                        IF temporalCounter_i1.done THEN 
                            (* Transition: '<S30>:42' *)
                            is_c47_ChiefMaster := ChiefMaster_IN_Error;
                            (* Entry 'Error': '<S30>:38' *)
                            (* '<S30>:38:2' MainHV_Minus_Welded = true *)
                            MainHV_Minus_Welded := TRUE;
                            (* '<S30>:38:3' MainHV_Plus_Welded = true *)
                            MainHV_Plus_Welded := TRUE;
                            (* '<S30>:38:4' WeldingDetection_Status = uint8(2); *)
                            WeldingDetection_Status := 2;
                        ELSE 
                            (* '<S30>:40:2' REQ_MainHV_ON_PLUS = false *)
                            REQ_MainHV_ON_PLUS := FALSE;
                            (* '<S30>:40:3' REQ_MainHV_ON_MINUS = false *)
                            REQ_MainHV_ON_MINUS := FALSE;
                            (* '<S30>:40:4' MainHV_Minus_Welded = false *)
                            MainHV_Minus_Welded := FALSE;
                            (* '<S30>:40:5' MainHV_Plus_Welded = false *)
                            MainHV_Plus_Welded := FALSE;
                        END_IF;

                    END_IF;

                ChiefMaster_IN_Open1: 
                    (* During 'Open1': '<S30>:28' *)
                    (* '<S30>:44:1' sf_internal_predicateOutput = In == true; *)

                    IF In THEN 
                        (* Transition: '<S30>:44' *)
                        is_c47_ChiefMaster := b_ChiefMaster_IN_Open;
                        temporalCounter_i1(timerAction := 1, maxTime := 0);
                        (* Entry 'Open': '<S30>:40' *)
                        (* '<S30>:40:2' REQ_MainHV_ON_PLUS = false *)
                        REQ_MainHV_ON_PLUS := FALSE;
                        (* '<S30>:40:3' REQ_MainHV_ON_MINUS = false *)
                        REQ_MainHV_ON_MINUS := FALSE;
                        (* '<S30>:40:4' MainHV_Minus_Welded = false *)
                        MainHV_Minus_Welded := FALSE;
                        (* '<S30>:40:5' MainHV_Plus_Welded = false *)
                        MainHV_Plus_Welded := FALSE;
                    ELSE 
                        (* '<S30>:28:2' REQ_MainHV_ON_PLUS = false *)
                        REQ_MainHV_ON_PLUS := FALSE;
                        (* '<S30>:28:3' REQ_MainHV_ON_MINUS = false *)
                        REQ_MainHV_ON_MINUS := FALSE;
                        (* '<S30>:28:4' MainHV_Minus_Welded = false *)
                        MainHV_Minus_Welded := FALSE;
                        (* '<S30>:28:5' MainHV_Plus_Welded = false *)
                        MainHV_Plus_Welded := FALSE;
                        (* '<S30>:28:6' WeldingDetection_Status = uint8(1); *)
                        WeldingDetection_Status := 1;
                    END_IF;

                ELSE
                    (* During 'Plus_Close': '<S30>:4' *)
                    (* '<S30>:13:1' sf_internal_predicateOutput = LoadVtg <= 20; *)

                    IF LoadVtg <= 20.0 THEN 
                        (* Transition: '<S30>:13' *)
                        is_c47_ChiefMaster := ChiefMaster_IN_Minus_Close;
                        temporalCounter_i1(timerAction := 1, maxTime := 0);
                        (* Entry 'Minus_Close': '<S30>:12' *)
                        (* '<S30>:12:2' REQ_MainHV_ON_MINUS = true *)
                        REQ_MainHV_ON_MINUS := TRUE;
                    ELSE 
                        (* '<S30>:23:1' sf_internal_predicateOutput = after(5,sec); *)
                        temporalCounter_i1(timerAction := 2, maxTime := 5000);

                        IF temporalCounter_i1.done THEN 
                            (* Transition: '<S30>:23' *)
                            is_c47_ChiefMaster := ChiefMaster_IN_ErrorMinus;
                            (* Entry 'ErrorMinus': '<S30>:22' *)
                            (* '<S30>:22:2' MainHV_Minus_Welded = true *)
                            MainHV_Minus_Welded := TRUE;
                            (* '<S30>:22:3' WeldingDetection_Status = uint8(2); *)
                            WeldingDetection_Status := 2;
                        ELSE 
                            (* '<S30>:4:2' REQ_MainHV_ON_PLUS = true *)
                            REQ_MainHV_ON_PLUS := TRUE;
                        END_IF;

                    END_IF;

            END_CASE;

        END_IF;

        (* End of Chart: '<S22>/Chart_WeldingDetection' *)
END_CASE;

END_FUNCTION_BLOCK

// Device/Application/Chart_jj
FUNCTION_BLOCK Chart_jj
VAR_INPUT
	ssMethodType: SINT;
	In: LREAL;
	b_n: LREAL;
END_VAR
VAR_OUTPUT
	Out: BOOL;
END_VAR
VAR
	temporalCounter_i1: PLC_CODER_TIMER;
	is_c10_ChiefMaster: USINT;
	is_active_c10_ChiefMaster: USINT;
END_VAR



CASE ssMethodType OF
    SS_INITIALIZE: 
        temporalCounter_i1(timerAction := 1, maxTime := 0);
        is_active_c10_ChiefMaster := 0;
        is_c10_ChiefMaster := ChiefMaster_IN_NO_ACTIVE_CHILD_a4;
        Out := FALSE;
    SS_OUTPUT: 
        (* Chart: '<S81>/Chart' *)
        (* Gateway: ChiefMaster/Flow Logic/Reset/Reset_Req/Subsystem1/Chart *)
        (* During: ChiefMaster/Flow Logic/Reset/Reset_Req/Subsystem1/Chart *)

        IF is_active_c10_ChiefMaster = 0 THEN 
            (* Entry: ChiefMaster/Flow Logic/Reset/Reset_Req/Subsystem1/Chart *)
            is_active_c10_ChiefMaster := 1;
            (* Entry Internal: ChiefMaster/Flow Logic/Reset/Reset_Req/Subsystem1/Chart *)
            (* Transition: '<S87>:3' *)
            is_c10_ChiefMaster := ChiefMaster_IN_Default_m;
            (* Entry 'Default': '<S87>:2' *)
            (* '<S87>:2:2' Out = false *)
            Out := FALSE;
        ELSE 

            CASE is_c10_ChiefMaster OF
                ChiefMaster_IN_Default_m: 
                    (* During 'Default': '<S87>:2' *)
                    (* '<S87>:6:1' sf_internal_predicateOutput = In == 2; *)

                    IF In = 2.0 THEN 
                        (* Transition: '<S87>:6' *)
                        is_c10_ChiefMaster := ChiefMaster_IN_Delay;
                        temporalCounter_i1(timerAction := 1, maxTime := 0);
                        (* Entry 'Delay': '<S87>:5' *)
                        (* '<S87>:5:2' Out = false *)
                        Out := FALSE;
                    ELSE 
                        (* '<S87>:2:2' Out = false *)
                        Out := FALSE;
                    END_IF;

                ChiefMaster_IN_Delay: 
                    (* During 'Delay': '<S87>:5' *)
                    (* '<S87>:12:1' sf_internal_predicateOutput = after(n,sec); *)
                    temporalCounter_i1(timerAction := 2, maxTime := TRUNC(b_n * 1000.0));

                    IF temporalCounter_i1.done THEN 
                        (* Transition: '<S87>:12' *)
                        is_c10_ChiefMaster := b_ChiefMaster_IN_Delay1;
                        (* Entry 'Delay1': '<S87>:11' *)
                        (* '<S87>:11:2' Out = true *)
                        Out := TRUE;
                    ELSE 
                        (* '<S87>:13:1' sf_internal_predicateOutput = In == 1 ||... *)
                        (* '<S87>:13:2' In == 3; *)

                        IF (In = 1.0) OR (In = 3.0) THEN 
                            (* Transition: '<S87>:13' *)
                            is_c10_ChiefMaster := ChiefMaster_IN_Default_m;
                            (* Entry 'Default': '<S87>:2' *)
                            (* '<S87>:2:2' Out = false *)
                            Out := FALSE;
                        ELSE 
                            (* '<S87>:5:2' Out = false *)
                            Out := FALSE;
                        END_IF;

                    END_IF;

                ELSE
                    (* During 'Delay1': '<S87>:11' *)
                    (* '<S87>:14:1' sf_internal_predicateOutput = In == 3; *)

                    IF In = 3.0 THEN 
                        (* Transition: '<S87>:14' *)
                        is_c10_ChiefMaster := ChiefMaster_IN_Default_m;
                        (* Entry 'Default': '<S87>:2' *)
                        (* '<S87>:2:2' Out = false *)
                        Out := FALSE;
                    ELSE 
                        (* '<S87>:11:2' Out = true *)
                        Out := TRUE;
                    END_IF;

            END_CASE;

        END_IF;

        (* End of Chart: '<S81>/Chart' *)
END_CASE;

END_FUNCTION_BLOCK

// Device/Application/Chart1
FUNCTION_BLOCK Chart1
VAR_INPUT
	ssMethodType: SINT;
	In: BOOL;
END_VAR
VAR_OUTPUT
	Out: BOOL;
END_VAR
VAR
	is_active_c12_ChiefMaster: USINT;
	is_c12_ChiefMaster: USINT;
	temporalCounter_i1: PLC_CODER_TIMER;
END_VAR



CASE ssMethodType OF
    SS_INITIALIZE: 
        temporalCounter_i1(timerAction := 1, maxTime := 0);
        is_active_c12_ChiefMaster := 0;
        is_c12_ChiefMaster := ChiefMaster_IN_NO_ACTIVE_CHILD_kt;
        Out := FALSE;
    SS_OUTPUT: 
        (* Chart: '<S81>/Chart1' *)
        (* Gateway: ChiefMaster/Flow Logic/Reset/Reset_Req/Subsystem1/Chart1 *)
        (* During: ChiefMaster/Flow Logic/Reset/Reset_Req/Subsystem1/Chart1 *)

        IF is_active_c12_ChiefMaster = 0 THEN 
            (* Entry: ChiefMaster/Flow Logic/Reset/Reset_Req/Subsystem1/Chart1 *)
            is_active_c12_ChiefMaster := 1;
            (* Entry Internal: ChiefMaster/Flow Logic/Reset/Reset_Req/Subsystem1/Chart1 *)
            (* Transition: '<S88>:3' *)
            is_c12_ChiefMaster := ChiefMaster_IN_Default_dh;
            (* Entry 'Default': '<S88>:2' *)
            (* '<S88>:2:2' Out = false *)
            Out := FALSE;
        ELSE 

            CASE is_c12_ChiefMaster OF
                ChiefMaster_IN_Default_dh: 
                    (* During 'Default': '<S88>:2' *)
                    (* '<S88>:6:1' sf_internal_predicateOutput = In == true; *)

                    IF In THEN 
                        (* Transition: '<S88>:6' *)
                        is_c12_ChiefMaster := ChiefMaster_IN_Delay_j;
                        temporalCounter_i1(timerAction := 1, maxTime := 0);
                        (* Entry 'Delay': '<S88>:5' *)
                        (* '<S88>:5:2' Out = true *)
                        Out := TRUE;
                    ELSE 
                        (* '<S88>:2:2' Out = false *)
                        Out := FALSE;
                    END_IF;

                ChiefMaster_IN_Delay_j: 
                    (* During 'Delay': '<S88>:5' *)
                    (* '<S88>:21:1' sf_internal_predicateOutput = after(10,msec); *)
                    temporalCounter_i1(timerAction := 2, maxTime := 10);

                    IF temporalCounter_i1.done THEN 
                        (* Transition: '<S88>:21' *)
                        is_c12_ChiefMaster := ChiefMaster_IN_pulse;
                        (* Entry 'pulse': '<S88>:20' *)
                        (* '<S88>:20:2' Out = false *)
                        Out := FALSE;
                    ELSE 
                        (* '<S88>:5:2' Out = true *)
                        Out := TRUE;
                    END_IF;

                ELSE
                    (* During 'pulse': '<S88>:20' *)
                    (* '<S88>:20:2' Out = false *)
                    Out := FALSE;
            END_CASE;

        END_IF;

        (* End of Chart: '<S81>/Chart1' *)
END_CASE;

END_FUNCTION_BLOCK

// Device/Application/Chart_lg
FUNCTION_BLOCK Chart_lg
VAR_INPUT
	ssMethodType: SINT;
	Error: BOOL;
	KL15_reset: BOOL;
END_VAR
VAR_OUTPUT
	SW_Reset: BOOL;
END_VAR
VAR
	temporalCounter_i1: PLC_CODER_TIMER;
	is_c13_ChiefMaster: USINT;
	is_active_c13_ChiefMaster: USINT;
END_VAR



CASE ssMethodType OF
    SS_INITIALIZE: 
        temporalCounter_i1(timerAction := 1, maxTime := 0);
        is_active_c13_ChiefMaster := 0;
        is_c13_ChiefMaster := ChiefMaster_IN_NO_ACTIVE_CHILD_a0;
        SW_Reset := FALSE;
    SS_OUTPUT: 
        (* Chart: '<S83>/Chart' *)
        (* Gateway: ChiefMaster/Flow Logic/Reset/Reset_Req/Subsystem3/Chart *)
        (* During: ChiefMaster/Flow Logic/Reset/Reset_Req/Subsystem3/Chart *)

        IF is_active_c13_ChiefMaster = 0 THEN 
            (* Entry: ChiefMaster/Flow Logic/Reset/Reset_Req/Subsystem3/Chart *)
            is_active_c13_ChiefMaster := 1;
            (* Entry Internal: ChiefMaster/Flow Logic/Reset/Reset_Req/Subsystem3/Chart *)
            (* Transition: '<S91>:3' *)
            is_c13_ChiefMaster := ChiefMaster_IN_Default_e0;
            (* Entry 'Default': '<S91>:2' *)
            (* '<S91>:2:2' SW_Reset = false *)
            SW_Reset := FALSE;
        ELSE 

            CASE is_c13_ChiefMaster OF
                ChiefMaster_IN_Default_e0: 
                    (* During 'Default': '<S91>:2' *)
                    (* '<S91>:6:1' sf_internal_predicateOutput = Error == true; *)

                    IF Error THEN 
                        (* Transition: '<S91>:6' *)
                        is_c13_ChiefMaster := ChiefMaster_IN_hold_hw;
                        temporalCounter_i1(timerAction := 1, maxTime := 0);
                        (* Entry 'hold': '<S91>:5' *)
                        (* '<S91>:5:2' SW_Reset = false *)
                        SW_Reset := FALSE;
                    ELSE 
                        (* '<S91>:2:2' SW_Reset = false *)
                        SW_Reset := FALSE;
                    END_IF;

                ChiefMaster_IN_Delay_i: 
                    (* During 'Delay': '<S91>:11' *)
                    (* '<S91>:16:1' sf_internal_predicateOutput = after(10,msec); *)
                    temporalCounter_i1(timerAction := 2, maxTime := 10);

                    IF temporalCounter_i1.done THEN 
                        (* Transition: '<S91>:16' *)
                        is_c13_ChiefMaster := ChiefMaster_IN_pulse_i;
                        (* Entry 'pulse': '<S91>:15' *)
                        (* '<S91>:15:2' SW_Reset = false *)
                        SW_Reset := FALSE;
                    ELSE 
                        (* '<S91>:11:2' SW_Reset = true *)
                        SW_Reset := TRUE;
                    END_IF;

                ChiefMaster_IN_KL15_reset: 
                    (* During 'KL15_reset': '<S91>:18' *)
                    (* '<S91>:21:1' sf_internal_predicateOutput = after(25,sec) &&... *)
                    (* '<S91>:21:2' Error == false; *)
                    temporalCounter_i1(timerAction := 2, maxTime := 25000);

                    IF temporalCounter_i1.done THEN 

                        IF  NOT Error THEN 
                            (* Transition: '<S91>:21' *)
                            is_c13_ChiefMaster := ChiefMaster_IN_Default_e0;
                            (* Entry 'Default': '<S91>:2' *)
                            (* '<S91>:2:2' SW_Reset = false *)
                            SW_Reset := FALSE;
                        ELSE 
                            (* '<S91>:18:2' SW_Reset = false *)
                            SW_Reset := FALSE;
                        END_IF;

                    ELSE 
                        (* '<S91>:18:2' SW_Reset = false *)
                        SW_Reset := FALSE;
                    END_IF;

                ChiefMaster_IN_hold_hw: 
                    (* During 'hold': '<S91>:5' *)
                    (* '<S91>:12:1' sf_internal_predicateOutput = after(5,sec); *)
                    temporalCounter_i1(timerAction := 2, maxTime := 5000);

                    IF temporalCounter_i1.done THEN 
                        (* Transition: '<S91>:12' *)
                        is_c13_ChiefMaster := ChiefMaster_IN_Delay_i;
                        temporalCounter_i1(timerAction := 1, maxTime := 0);
                        (* Entry 'Delay': '<S91>:11' *)
                        (* '<S91>:11:2' SW_Reset = true *)
                        SW_Reset := TRUE;
                    ELSE 
                        (* '<S91>:13:1' sf_internal_predicateOutput = Error == false; *)

                        IF  NOT Error THEN 
                            (* Transition: '<S91>:13' *)
                            is_c13_ChiefMaster := ChiefMaster_IN_Default_e0;
                            (* Entry 'Default': '<S91>:2' *)
                            (* '<S91>:2:2' SW_Reset = false *)
                            SW_Reset := FALSE;
                        ELSE 
                            (* '<S91>:5:2' SW_Reset = false *)
                            SW_Reset := FALSE;
                        END_IF;

                    END_IF;

                ELSE
                    (* During 'pulse': '<S91>:15' *)
                    (* '<S91>:17:1' sf_internal_predicateOutput = KL15_reset == true; *)

                    IF KL15_reset THEN 
                        (* Transition: '<S91>:17' *)
                        is_c13_ChiefMaster := ChiefMaster_IN_KL15_reset;
                        temporalCounter_i1(timerAction := 1, maxTime := 0);
                        (* Entry 'KL15_reset': '<S91>:18' *)
                        (* '<S91>:18:2' SW_Reset = false *)
                        SW_Reset := FALSE;
                    ELSE 
                        (* '<S91>:15:2' SW_Reset = false *)
                        SW_Reset := FALSE;
                    END_IF;

            END_CASE;

        END_IF;

        (* End of Chart: '<S83>/Chart' *)
END_CASE;

END_FUNCTION_BLOCK

// Device/Application/Chart1_l
FUNCTION_BLOCK Chart1_l
VAR_INPUT
	ssMethodType: SINT;
	SW_Reset: BOOL;
	KL_15_reset_CM: BOOL;
END_VAR
VAR_OUTPUT
	Count: LREAL;
END_VAR
VAR
	is_active_c14_ChiefMaster: USINT;
	is_c14_ChiefMaster: USINT;
END_VAR



CASE ssMethodType OF
    SS_INITIALIZE: 
        is_active_c14_ChiefMaster := 0;
        is_c14_ChiefMaster := ChiefMaster_IN_NO_ACTIVE_CHILD_a1;
        Count := 0.0;
    SS_OUTPUT: 
        (* Chart: '<S83>/Chart1' *)
        (* Gateway: ChiefMaster/Flow Logic/Reset/Reset_Req/Subsystem3/Chart1 *)
        (* During: ChiefMaster/Flow Logic/Reset/Reset_Req/Subsystem3/Chart1 *)

        IF is_active_c14_ChiefMaster = 0 THEN 
            (* Entry: ChiefMaster/Flow Logic/Reset/Reset_Req/Subsystem3/Chart1 *)
            is_active_c14_ChiefMaster := 1;
            (* Entry Internal: ChiefMaster/Flow Logic/Reset/Reset_Req/Subsystem3/Chart1 *)
            (* Transition: '<S92>:3' *)
            is_c14_ChiefMaster := ChiefMaster_IN_Default_g;
            (* Entry 'Default': '<S92>:2' *)
            (* '<S92>:2:2' Count = 0 *)
            Count := 0.0;
        ELSE 

            CASE is_c14_ChiefMaster OF
                ChiefMaster_IN_Default_g: 
                    (* During 'Default': '<S92>:2' *)
                    (* '<S92>:6:1' sf_internal_predicateOutput = SW_Reset == true; *)

                    IF SW_Reset THEN 
                        (* Transition: '<S92>:6' *)
                        is_c14_ChiefMaster := ChiefMaster_IN_Delay_m;
                        (* Entry 'Delay': '<S92>:5' *)
                        (* '<S92>:5:2' Count = Count + 1 *)
                        Count := Count + 1.0;
                    ELSE 
                        (* '<S92>:2:2' Count = 0 *)
                        Count := 0.0;
                    END_IF;

                ChiefMaster_IN_Delay_m: 
                    (* During 'Delay': '<S92>:5' *)
                    (* '<S92>:28:1' sf_internal_predicateOutput = SW_Reset == false; *)

                    IF  NOT SW_Reset THEN 
                        (* Transition: '<S92>:28' *)
                        is_c14_ChiefMaster := ChiefMaster_IN_Delay1_h;
                        (* Entry 'Delay1': '<S92>:27' *)
                    ELSE 
                        (* '<S92>:5:2' Count = Count + 1 *)
                        Count := Count + 1.0;
                    END_IF;

                ELSE
                    (* During 'Delay1': '<S92>:27' *)
                    (* '<S92>:24:1' sf_internal_predicateOutput = KL_15_reset_CM == true; *)

                    IF KL_15_reset_CM THEN 
                        (* Transition: '<S92>:24' *)
                        is_c14_ChiefMaster := ChiefMaster_IN_Default_g;
                        (* Entry 'Default': '<S92>:2' *)
                        (* '<S92>:2:2' Count = 0 *)
                        Count := 0.0;
                    ELSE 
                        (* '<S92>:29:1' sf_internal_predicateOutput = SW_Reset == true; *)

                        IF SW_Reset THEN 
                            (* Transition: '<S92>:29' *)
                            is_c14_ChiefMaster := ChiefMaster_IN_Delay_m;
                            (* Entry 'Delay': '<S92>:5' *)
                            (* '<S92>:5:2' Count = Count + 1 *)
                            Count := Count + 1.0;
                        END_IF;

                    END_IF;

            END_CASE;

        END_IF;

        (* End of Chart: '<S83>/Chart1' *)
END_CASE;

END_FUNCTION_BLOCK

// Device/Application/CMState
FUNCTION_BLOCK CMState
VAR_INPUT
	ssMethodType: SINT;
	KL15: BOOL;
	KL15_AllBoxes: BOOL;
	InsulationReadyOK: BOOL;
	BattRelay_Closed: BOOL;
	IMD_Available: BOOL;
	BattRelay_Close_Req: BOOL;
	REQ_IMD_ON: BOOL;
	FL_boREQ_MainHV_ON_MINUS: BOOL;
	MainHV_Plus_Status: LREAL;
	ShutdownError: BOOL;
END_VAR
VAR_OUTPUT
	FL_u8SS_ChiefMaster_State: USINT;
END_VAR
VAR
	is_c27_ChiefMaster: USINT;
	is_active_c27_ChiefMaster: USINT;
	is_ON: USINT;
	is_OFF: USINT;
	tmp: BOOL;
END_VAR



CASE ssMethodType OF
    SS_INITIALIZE: 
        (* SystemInitialize for Chart: '<S109>/CMState' *)
        is_OFF := ChiefMaster_IN_NO_ACTIVE_CHILD_ktp;
        is_ON := ChiefMaster_IN_NO_ACTIVE_CHILD_ktp;
        is_active_c27_ChiefMaster := 0;
        is_c27_ChiefMaster := ChiefMaster_IN_NO_ACTIVE_CHILD_ktp;
        FL_u8SS_ChiefMaster_State := 0;
    SS_OUTPUT: 
        (* Chart: '<S109>/CMState' *)
        (* Gateway: ChiefMaster/Flow Logic/System Status/CMState/CMState *)
        (* During: ChiefMaster/Flow Logic/System Status/CMState/CMState *)

        IF is_active_c27_ChiefMaster = 0 THEN 
            (* Entry: ChiefMaster/Flow Logic/System Status/CMState/CMState *)
            is_active_c27_ChiefMaster := 1;
            (* Entry Internal: ChiefMaster/Flow Logic/System Status/CMState/CMState *)
            (* Transition: '<S124>:2' *)
            is_c27_ChiefMaster := ChiefMaster_IN_Sleep;
            (* Entry 'Sleep': '<S124>:1' *)
            (* '<S124>:1:2' CMState=0; *)
            FL_u8SS_ChiefMaster_State := 0;
        ELSE 

            CASE is_c27_ChiefMaster OF
                ChiefMaster_IN_Error_o: 
                    (* During 'Error': '<S124>:99' *)
                    (* '<S124>:116:1' sf_internal_predicateOutput = ShutdownError == false &&... *)
                    (* '<S124>:116:2' KL15==true; *)
                    tmp :=  NOT ShutdownError;

                    IF tmp AND KL15 THEN 
                        (* Transition: '<S124>:116' *)
                        is_c27_ChiefMaster := ChiefMaster_IN_ON;
                        (* Entry Internal 'ON': '<S124>:31' *)
                        (* Transition: '<S124>:62' *)
                        is_ON := ChiefMaster_IN_KL15ON;
                        (* Entry 'KL15ON': '<S124>:3' *)
                        (* '<S124>:3:2' CMState=1; *)
                        FL_u8SS_ChiefMaster_State := 1;
                    ELSE 
                        (* '<S124>:117:1' sf_internal_predicateOutput = ShutdownError == false &&... *)
                        (* '<S124>:117:2' KL15==false; *)

                        IF tmp AND ( NOT KL15) THEN 
                            (* Transition: '<S124>:117' *)
                            is_c27_ChiefMaster := ChiefMaster_IN_OFF;
                            (* Entry Internal 'OFF': '<S124>:90' *)
                            (* Transition: '<S124>:92' *)
                            is_OFF := ChiefMaster_IN_BDURelayOpen_Req;
                            (* Entry 'BDURelayOpen_Req': '<S124>:82' *)
                            (* '<S124>:82:2' CMState=8; *)
                            FL_u8SS_ChiefMaster_State := 8;
                        ELSE 
                            (* '<S124>:99:2' CMState=14; *)
                            FL_u8SS_ChiefMaster_State := 14;
                        END_IF;

                    END_IF;

                ChiefMaster_IN_OFF: 
                    (* During 'OFF': '<S124>:90' *)
                    (* '<S124>:96:1' sf_internal_predicateOutput = CMState==13; *)

                    IF FL_u8SS_ChiefMaster_State = 13 THEN 
                        (* Transition: '<S124>:96' *)
                        (* Exit Internal 'OFF': '<S124>:90' *)
                        is_OFF := ChiefMaster_IN_NO_ACTIVE_CHILD_ktp;
                        is_c27_ChiefMaster := ChiefMaster_IN_Sleep;
                        (* Entry 'Sleep': '<S124>:1' *)
                        (* '<S124>:1:2' CMState=0; *)
                        FL_u8SS_ChiefMaster_State := 0;
                    ELSE 
                        (* '<S124>:100:1' sf_internal_predicateOutput = ShutdownError == true; *)

                        IF ShutdownError THEN 
                            (* Transition: '<S124>:100' *)
                            (* Exit Internal 'OFF': '<S124>:90' *)
                            is_OFF := ChiefMaster_IN_NO_ACTIVE_CHILD_ktp;
                            is_c27_ChiefMaster := ChiefMaster_IN_Error_o;
                            (* Entry 'Error': '<S124>:99' *)
                            (* '<S124>:99:2' CMState=14; *)
                            FL_u8SS_ChiefMaster_State := 14;
                        ELSE 

                            CASE is_OFF OF
                                ChiefMaster_IN_BDURelayOpen: 
                                    (* During 'BDURelayOpen': '<S124>:86' *)
                                    (* '<S124>:84:1' sf_internal_predicateOutput = BattRelay_Close_Req==false; *)

                                    IF  NOT BattRelay_Close_Req THEN 
                                        (* Transition: '<S124>:84' *)
                                        is_OFF := ChiefMaster_IN_BattRelayOpen_Req;
                                        (* Entry 'BattRelayOpen_Req': '<S124>:94' *)
                                        (* '<S124>:94:2' CMState=10; *)
                                        FL_u8SS_ChiefMaster_State := 10;
                                    ELSE 
                                        (* '<S124>:86:2' CMState=9; *)
                                        FL_u8SS_ChiefMaster_State := 9;
                                    END_IF;

                                ChiefMaster_IN_BDURelayOpen_Req: 
                                    (* During 'BDURelayOpen_Req': '<S124>:82' *)
                                    (* '<S124>:93:1' sf_internal_predicateOutput = MainHV_Plus_Status==0; *)

                                    IF MainHV_Plus_Status = 0.0 THEN 
                                        (* Transition: '<S124>:93' *)
                                        is_OFF := ChiefMaster_IN_BDURelayOpen;
                                        (* Entry 'BDURelayOpen': '<S124>:86' *)
                                        (* '<S124>:86:2' CMState=9; *)
                                        FL_u8SS_ChiefMaster_State := 9;
                                    ELSE 
                                        (* '<S124>:82:2' CMState=8; *)
                                        FL_u8SS_ChiefMaster_State := 8;
                                    END_IF;

                                ChiefMaster_IN_BattRelayOpen: 
                                    (* During 'BattRelayOpen': '<S124>:89' *)
                                    (* '<S124>:83:1' sf_internal_predicateOutput = REQ_IMD_ON == false; *)

                                    IF  NOT REQ_IMD_ON THEN 
                                        (* Transition: '<S124>:83' *)
                                        is_OFF := ChiefMaster_IN_ISOMonitorOFF;
                                        (* Entry 'ISOMonitorOFF': '<S124>:88' *)
                                        (* '<S124>:88:2' CMState=12; *)
                                        FL_u8SS_ChiefMaster_State := 12;
                                    ELSE 
                                        (* '<S124>:89:2' CMState=11; *)
                                        FL_u8SS_ChiefMaster_State := 11;
                                    END_IF;

                                ChiefMaster_IN_BattRelayOpen_Req: 
                                    (* During 'BattRelayOpen_Req': '<S124>:94' *)
                                    (* '<S124>:95:1' sf_internal_predicateOutput = BattRelay_Closed==false; *)

                                    IF  NOT BattRelay_Closed THEN 
                                        (* Transition: '<S124>:95' *)
                                        is_OFF := ChiefMaster_IN_BattRelayOpen;
                                        (* Entry 'BattRelayOpen': '<S124>:89' *)
                                        (* '<S124>:89:2' CMState=11; *)
                                        FL_u8SS_ChiefMaster_State := 11;
                                    ELSE 
                                        (* '<S124>:94:2' CMState=10; *)
                                        FL_u8SS_ChiefMaster_State := 10;
                                    END_IF;

                                ChiefMaster_IN_ISOMonitorOFF: 
                                    (* During 'ISOMonitorOFF': '<S124>:88' *)
                                    (* '<S124>:85:1' sf_internal_predicateOutput = KL15_AllBoxes==false; *)

                                    IF  NOT KL15_AllBoxes THEN 
                                        (* Transition: '<S124>:85' *)
                                        is_OFF := ChiefMaster_IN_KL15OFF;
                                        (* Entry 'KL15OFF': '<S124>:91' *)
                                        (* '<S124>:91:2' CMState=13; *)
                                        FL_u8SS_ChiefMaster_State := 13;
                                    ELSE 
                                        (* '<S124>:88:2' CMState=12; *)
                                        FL_u8SS_ChiefMaster_State := 12;
                                    END_IF;

                                ELSE
                                    (* During 'KL15OFF': '<S124>:91' *)
                                    (* '<S124>:91:2' CMState=13; *)
                                    FL_u8SS_ChiefMaster_State := 13;
                            END_CASE;

                        END_IF;

                    END_IF;

                ChiefMaster_IN_ON: 
                    (* During 'ON': '<S124>:31' *)
                    (* '<S124>:87:1' sf_internal_predicateOutput = KL15==false; *)

                    IF  NOT KL15 THEN 
                        (* Transition: '<S124>:87' *)
                        (* Exit Internal 'ON': '<S124>:31' *)
                        is_ON := ChiefMaster_IN_NO_ACTIVE_CHILD_ktp;
                        is_c27_ChiefMaster := ChiefMaster_IN_OFF;
                        (* Entry Internal 'OFF': '<S124>:90' *)
                        (* Transition: '<S124>:92' *)
                        is_OFF := ChiefMaster_IN_BDURelayOpen_Req;
                        (* Entry 'BDURelayOpen_Req': '<S124>:82' *)
                        (* '<S124>:82:2' CMState=8; *)
                        FL_u8SS_ChiefMaster_State := 8;
                    ELSE 
                        (* '<S124>:101:1' sf_internal_predicateOutput = ShutdownError == true; *)

                        IF ShutdownError THEN 
                            (* Transition: '<S124>:101' *)
                            (* Exit Internal 'ON': '<S124>:31' *)
                            is_ON := ChiefMaster_IN_NO_ACTIVE_CHILD_ktp;
                            is_c27_ChiefMaster := ChiefMaster_IN_Error_o;
                            (* Entry 'Error': '<S124>:99' *)
                            (* '<S124>:99:2' CMState=14; *)
                            FL_u8SS_ChiefMaster_State := 14;
                        ELSE 

                            CASE is_ON OF
                                ChiefMaster_IN_BDURelayClose: 
                                    (* During 'BDURelayClose': '<S124>:73' *)
                                    (* '<S124>:73:2' CMState=7; *)
                                    FL_u8SS_ChiefMaster_State := 7;
                                ChiefMaster_IN_BDURelayClose_Req: 
                                    (* During 'BDURelayClose_Req': '<S124>:19' *)
                                    (* '<S124>:74:1' sf_internal_predicateOutput = MainHV_Plus_Status == 2; *)

                                    IF MainHV_Plus_Status = 2.0 THEN 
                                        (* Transition: '<S124>:74' *)
                                        is_ON := ChiefMaster_IN_BDURelayClose;
                                        (* Entry 'BDURelayClose': '<S124>:73' *)
                                        (* '<S124>:73:2' CMState=7; *)
                                        FL_u8SS_ChiefMaster_State := 7;
                                    ELSE 
                                        (* '<S124>:19:2' CMState=6; *)
                                        FL_u8SS_ChiefMaster_State := 6;
                                    END_IF;

                                ChiefMaster_IN_BattRelayClose: 
                                    (* During 'BattRelayClose': '<S124>:16' *)
                                    (* '<S124>:68:1' sf_internal_predicateOutput = FL_boREQ_MainHV_ON_MINUS == true; *)

                                    IF FL_boREQ_MainHV_ON_MINUS THEN 
                                        (* Transition: '<S124>:68' *)
                                        is_ON := ChiefMaster_IN_BDURelayClose_Req;
                                        (* Entry 'BDURelayClose_Req': '<S124>:19' *)
                                        (* '<S124>:19:2' CMState=6; *)
                                        FL_u8SS_ChiefMaster_State := 6;
                                    ELSE 
                                        (* '<S124>:71:1' sf_internal_predicateOutput = BattRelay_Closed==false; *)

                                        IF  NOT BattRelay_Closed THEN 
                                            (* Transition: '<S124>:71' *)
                                            is_ON := ChiefMaster_IN_BattRelayClose_Req;
                                            (* Entry 'BattRelayClose_Req': '<S124>:69' *)
                                            (* '<S124>:69:2' CMState=4; *)
                                            FL_u8SS_ChiefMaster_State := 4;
                                        ELSE 
                                            (* '<S124>:16:2' CMState=5; *)
                                            FL_u8SS_ChiefMaster_State := 5;
                                        END_IF;

                                    END_IF;

                                ChiefMaster_IN_BattRelayClose_Req: 
                                    (* During 'BattRelayClose_Req': '<S124>:69' *)
                                    (* '<S124>:70:1' sf_internal_predicateOutput = BattRelay_Closed==true; *)

                                    IF BattRelay_Closed THEN 
                                        (* Transition: '<S124>:70' *)
                                        is_ON := ChiefMaster_IN_BattRelayClose;
                                        (* Entry 'BattRelayClose': '<S124>:16' *)
                                        (* '<S124>:16:2' CMState=5; *)
                                        FL_u8SS_ChiefMaster_State := 5;
                                    ELSE 
                                        (* '<S124>:69:2' CMState=4; *)
                                        FL_u8SS_ChiefMaster_State := 4;
                                    END_IF;

                                ChiefMaster_IN_ISOMonitor_OK: 
                                    (* During 'ISOMonitor_OK': '<S124>:111' *)
                                    (* '<S124>:112:1' sf_internal_predicateOutput = BattRelay_Close_Req==true; *)

                                    IF BattRelay_Close_Req THEN 
                                        (* Transition: '<S124>:112' *)
                                        is_ON := ChiefMaster_IN_BattRelayClose_Req;
                                        (* Entry 'BattRelayClose_Req': '<S124>:69' *)
                                        (* '<S124>:69:2' CMState=4; *)
                                        FL_u8SS_ChiefMaster_State := 4;
                                    ELSE 
                                        (* '<S124>:111:2' CMState=3; *)
                                        FL_u8SS_ChiefMaster_State := 3;
                                    END_IF;

                                ChiefMaster_IN_ISOMonitor_check: 
                                    (* During 'ISOMonitor_check': '<S124>:13' *)
                                    (* '<S124>:17:1' sf_internal_predicateOutput = InsulationReadyOK==true; *)

                                    IF InsulationReadyOK THEN 
                                        (* Transition: '<S124>:17' *)
                                        is_ON := ChiefMaster_IN_ISOMonitor_OK;
                                        (* Entry 'ISOMonitor_OK': '<S124>:111' *)
                                        (* '<S124>:111:2' CMState=3; *)
                                        FL_u8SS_ChiefMaster_State := 3;
                                    ELSE 
                                        (* '<S124>:13:2' CMState=2; *)
                                        FL_u8SS_ChiefMaster_State := 2;
                                    END_IF;

                                ELSE
                                    (* During 'KL15ON': '<S124>:3' *)
                                    (* '<S124>:11:1' sf_internal_predicateOutput = KL15_AllBoxes==true && IMD_Available == true; *)

                                    IF KL15_AllBoxes AND IMD_Available THEN 
                                        (* Transition: '<S124>:11' *)
                                        is_ON := ChiefMaster_IN_ISOMonitor_check;
                                        (* Entry 'ISOMonitor_check': '<S124>:13' *)
                                        (* '<S124>:13:2' CMState=2; *)
                                        FL_u8SS_ChiefMaster_State := 2;
                                    ELSE 
                                        (* '<S124>:3:2' CMState=1; *)
                                        FL_u8SS_ChiefMaster_State := 1;
                                    END_IF;

                            END_CASE;

                        END_IF;

                    END_IF;

                ELSE
                    (* During 'Sleep': '<S124>:1' *)
                    (* '<S124>:4:1' sf_internal_predicateOutput = KL15==true; *)

                    IF KL15 THEN 
                        (* Transition: '<S124>:4' *)
                        is_c27_ChiefMaster := ChiefMaster_IN_ON;
                        (* Entry Internal 'ON': '<S124>:31' *)
                        (* Transition: '<S124>:62' *)
                        is_ON := ChiefMaster_IN_KL15ON;
                        (* Entry 'KL15ON': '<S124>:3' *)
                        (* '<S124>:3:2' CMState=1; *)
                        FL_u8SS_ChiefMaster_State := 1;
                    ELSE 
                        (* '<S124>:1:2' CMState=0; *)
                        FL_u8SS_ChiefMaster_State := 0;
                    END_IF;

            END_CASE;

        END_IF;

        (* End of Chart: '<S109>/CMState' *)
END_CASE;

END_FUNCTION_BLOCK

// Device/Application/EMSRET_Power
FUNCTION_BLOCK EMSRET_Power
VAR_INPUT
	ssMethodType: SINT;
	ESD: BOOL;
	HVILNOK: BOOL;
	b_Reset: BOOL;
END_VAR
VAR_OUTPUT
	FL_boSS_EMSRET_POWER: BOOL;
END_VAR
VAR
	i0_EMSRET: EMSRET;
	rtb_FL_boSS_EMSRET_POWER: BOOL;
END_VAR



CASE ssMethodType OF
    SS_INITIALIZE: 
        i0_EMSRET(ssMethodType := SS_INITIALIZE, AllOK := rtb_FL_boSS_EMSRET_POWER, b_Reset := b_Reset);
        FL_boSS_EMSRET_POWER := i0_EMSRET.EMSRET_mb;
    SS_OUTPUT: 
        (* Logic: '<S111>/AND' incorporates:
         *  Logic: '<S111>/NOT'
         *  Logic: '<S111>/NOT1' *)
        i0_EMSRET(ssMethodType := SS_OUTPUT, AllOK := ( NOT ESD) AND ( NOT HVILNOK), b_Reset := b_Reset);
        FL_boSS_EMSRET_POWER := i0_EMSRET.EMSRET_mb;
END_CASE;

END_FUNCTION_BLOCK

// Device/Application/EMSRET
FUNCTION_BLOCK EMSRET
VAR_INPUT
	ssMethodType: SINT;
	AllOK: BOOL;
	b_Reset: BOOL;
END_VAR
VAR_OUTPUT
	EMSRET_mb: BOOL;
END_VAR
VAR
	is_active_c50_ChiefMaster: USINT;
	is_c50_ChiefMaster: USINT;
	temporalCounter_i1: PLC_CODER_TIMER;
END_VAR



CASE ssMethodType OF
    SS_INITIALIZE: 
        temporalCounter_i1(timerAction := 1, maxTime := 0);
        is_active_c50_ChiefMaster := 0;
        is_c50_ChiefMaster := ChiefMaster_IN_NO_ACTIVE_CHILD_jr;
        EMSRET_mb := FALSE;
    SS_OUTPUT: 
        (* Chart: '<S111>/EMSRET' *)
        (* Gateway: ChiefMaster/Flow Logic/System Status/EMSRET_Power/EMSRET *)
        (* During: ChiefMaster/Flow Logic/System Status/EMSRET_Power/EMSRET *)

        IF is_active_c50_ChiefMaster = 0 THEN 
            (* Entry: ChiefMaster/Flow Logic/System Status/EMSRET_Power/EMSRET *)
            is_active_c50_ChiefMaster := 1;
            (* Entry Internal: ChiefMaster/Flow Logic/System Status/EMSRET_Power/EMSRET *)
            (* Transition: '<S138>:2' *)
            is_c50_ChiefMaster := ChiefMaster_IN_OFF_i;
            (* Entry 'OFF': '<S138>:1' *)
            (* '<S138>:1:2' EMSRET=false; *)
            EMSRET_mb := FALSE;
        ELSE 

            CASE is_c50_ChiefMaster OF
                ChiefMaster_IN_Delay_b: 
                    (* During 'Delay': '<S138>:8' *)
                    (* '<S138>:13:1' sf_internal_predicateOutput = after(3,sec); *)
                    temporalCounter_i1(timerAction := 2, maxTime := 3000);

                    IF temporalCounter_i1.done THEN 
                        (* Transition: '<S138>:13' *)
                        is_c50_ChiefMaster := ChiefMaster_IN_ShutOff;
                        (* Entry 'ShutOff': '<S138>:12' *)
                        (* '<S138>:12:2' EMSRET=false; *)
                        EMSRET_mb := FALSE;
                    ELSE 
                        (* '<S138>:8:2' EMSRET=true; *)
                        EMSRET_mb := TRUE;
                    END_IF;

                ChiefMaster_IN_OFF_i: 
                    (* During 'OFF': '<S138>:1' *)
                    (* '<S138>:6:1' sf_internal_predicateOutput = AllOK==true; *)

                    IF AllOK THEN 
                        (* Transition: '<S138>:6' *)
                        is_c50_ChiefMaster := ChiefMaster_IN_ON_g;
                        (* Entry 'ON': '<S138>:5' *)
                        (* '<S138>:5:2' EMSRET=true; *)
                        EMSRET_mb := TRUE;
                    ELSE 
                        (* '<S138>:1:2' EMSRET=false; *)
                        EMSRET_mb := FALSE;
                    END_IF;

                ChiefMaster_IN_ON_g: 
                    (* During 'ON': '<S138>:5' *)
                    (* '<S138>:10:1' sf_internal_predicateOutput = AllOK==false; *)

                    IF  NOT AllOK THEN 
                        (* Transition: '<S138>:10' *)
                        is_c50_ChiefMaster := ChiefMaster_IN_Delay_b;
                        temporalCounter_i1(timerAction := 1, maxTime := 0);
                        (* Entry 'Delay': '<S138>:8' *)
                        (* '<S138>:8:2' EMSRET=true; *)
                        EMSRET_mb := TRUE;
                    ELSE 
                        (* '<S138>:5:2' EMSRET=true; *)
                        EMSRET_mb := TRUE;
                    END_IF;

                ELSE
                    (* During 'ShutOff': '<S138>:12' *)
                    (* '<S138>:15:1' sf_internal_predicateOutput = Reset==true; *)

                    IF b_Reset THEN 
                        (* Transition: '<S138>:15' *)
                        is_c50_ChiefMaster := ChiefMaster_IN_OFF_i;
                        (* Entry 'OFF': '<S138>:1' *)
                        (* '<S138>:1:2' EMSRET=false; *)
                        EMSRET_mb := FALSE;
                    ELSE 
                        (* '<S138>:12:2' EMSRET=false; *)
                        EMSRET_mb := FALSE;
                    END_IF;

            END_CASE;

        END_IF;

        (* End of Chart: '<S111>/EMSRET' *)
END_CASE;

END_FUNCTION_BLOCK

// Device/Application/Chart_Hysteresis_HighActive
FUNCTION_BLOCK Chart_Hysteresis_HighActive
VAR_INPUT
	ssMethodType: SINT;
	sSignal: REAL;
	boInitial_Value: BOOL;
	boValue_Activated: BOOL;
	boValue_Deactivated: BOOL;
	sLB: REAL;
	b_sUB: REAL;
END_VAR
VAR_OUTPUT
	boOutput: BOOL;
END_VAR
VAR
	is_active_c1_Library_DataProcessing_v1_1: USINT;
	is_c1_Library_DataProcessing_v1_1: USINT;
END_VAR



CASE ssMethodType OF
    SS_INITIALIZE: 
        is_active_c1_Library_DataProcessing_v1_1 := 0;
        is_c1_Library_DataProcessing_v1_1 := ChiefMaster_IN_NO_ACTIVE_CHILD_p;
        boOutput := FALSE;
    SS_OUTPUT: 
        (* Chart: '<S395>/Chart_Hysteresis_HighActive' *)
        (* Gateway: Lib_Hysteresis_HighActive/Chart_Hysteresis_HighActive *)
        (* During: Lib_Hysteresis_HighActive/Chart_Hysteresis_HighActive *)

        IF is_active_c1_Library_DataProcessing_v1_1 = 0 THEN 
            (* Entry: Lib_Hysteresis_HighActive/Chart_Hysteresis_HighActive *)
            is_active_c1_Library_DataProcessing_v1_1 := 1;
            (* Entry Internal: Lib_Hysteresis_HighActive/Chart_Hysteresis_HighActive *)
            (* Transition: '<S396>:5' *)
            is_c1_Library_DataProcessing_v1_1 := ChiefMaster_IN_OFF_c;
            (* Entry 'OFF': '<S396>:8' *)
            (* '<S396>:8:3' boOutput= boInitial_Value; *)
            boOutput := boInitial_Value;
        ELSE 

            CASE is_c1_Library_DataProcessing_v1_1 OF
                ChiefMaster_IN_HighValue: 
                    (* During 'HighValue': '<S396>:4' *)
                    (* '<S396>:1:1' sf_internal_predicateOutput = sSignal<sLB; *)

                    IF sSignal < sLB THEN 
                        (* Transition: '<S396>:1' *)
                        is_c1_Library_DataProcessing_v1_1 := ChiefMaster_IN_LowValue;
                        (* Entry 'LowValue': '<S396>:2' *)
                        (* '<S396>:2:3' boOutput = boValue_Deactivated; *)
                        boOutput := boValue_Deactivated;
                    END_IF;

                ChiefMaster_IN_LowValue: 
                    (* During 'LowValue': '<S396>:2' *)
                    (* '<S396>:7:1' sf_internal_predicateOutput = sSignal>sUB; *)

                    IF sSignal > b_sUB THEN 
                        (* Transition: '<S396>:7' *)
                        is_c1_Library_DataProcessing_v1_1 := ChiefMaster_IN_HighValue;
                        (* Entry 'HighValue': '<S396>:4' *)
                        (* '<S396>:4:3' boOutput = boValue_Activated; *)
                        boOutput := boValue_Activated;
                    END_IF;

                ELSE
                    (* During 'OFF': '<S396>:8' *)
                    (* '<S396>:6:1' sf_internal_predicateOutput = sSignal<sLB; *)

                    IF sSignal < sLB THEN 
                        (* Transition: '<S396>:6' *)
                        is_c1_Library_DataProcessing_v1_1 := ChiefMaster_IN_LowValue;
                        (* Entry 'LowValue': '<S396>:2' *)
                        (* '<S396>:2:3' boOutput = boValue_Deactivated; *)
                        boOutput := boValue_Deactivated;
                    ELSE 
                        (* '<S396>:3:1' sf_internal_predicateOutput = sSignal>sUB; *)

                        IF sSignal > b_sUB THEN 
                            (* Transition: '<S396>:3' *)
                            is_c1_Library_DataProcessing_v1_1 := ChiefMaster_IN_HighValue;
                            (* Entry 'HighValue': '<S396>:4' *)
                            (* '<S396>:4:3' boOutput = boValue_Activated; *)
                            boOutput := boValue_Activated;
                        END_IF;

                    END_IF;

            END_CASE;

        END_IF;

        (* End of Chart: '<S395>/Chart_Hysteresis_HighActive' *)
END_CASE;

END_FUNCTION_BLOCK

// Device/Application/IMDOK_Input_Delay
FUNCTION_BLOCK IMDOK_Input_Delay
VAR_INPUT
	ssMethodType: SINT;
	In: BOOL;
END_VAR
VAR_OUTPUT
	out: BOOL;
END_VAR
VAR
	is_active_c59_ChiefMaster: USINT;
	is_c59_ChiefMaster: USINT;
	temporalCounter_i1: PLC_CODER_TIMER;
END_VAR



CASE ssMethodType OF
    SS_INITIALIZE: 
        temporalCounter_i1(timerAction := 1, maxTime := 0);
        is_active_c59_ChiefMaster := 0;
        is_c59_ChiefMaster := ChiefMaster_IN_NO_ACTIVE_CHILD_jg;
        out := FALSE;
    SS_OUTPUT: 
        (* Chart: '<S702>/IMDOK_Input_Delay' *)
        (* Gateway: ChiefMaster/Input Translation/Battery Signals/BatteryPackSignals/Subsystem4/IMDOK_Input_Delay *)
        (* During: ChiefMaster/Input Translation/Battery Signals/BatteryPackSignals/Subsystem4/IMDOK_Input_Delay *)

        IF is_active_c59_ChiefMaster = 0 THEN 
            (* Entry: ChiefMaster/Input Translation/Battery Signals/BatteryPackSignals/Subsystem4/IMDOK_Input_Delay *)
            is_active_c59_ChiefMaster := 1;
            (* Entry Internal: ChiefMaster/Input Translation/Battery Signals/BatteryPackSignals/Subsystem4/IMDOK_Input_Delay *)
            (* Transition: '<S706>:16' *)
            is_c59_ChiefMaster := ChiefMaster_IN_Initial1;
            temporalCounter_i1(timerAction := 1, maxTime := 0);
            (* Entry 'Initial1': '<S706>:20' *)
            (* '<S706>:20:3' out = false; *)
            out := FALSE;
        ELSE 

            CASE is_c59_ChiefMaster OF
                ChiefMaster_IN_After_delay1: 
                    (* During 'After_delay1': '<S706>:18' *)
                    (* '<S706>:18:3' out = In; *)
                    out := In;
                ELSE
                    (* During 'Initial1': '<S706>:20' *)
                    (* '<S706>:15:1' sf_internal_predicateOutput = after(7,sec); *)
                    temporalCounter_i1(timerAction := 2, maxTime := 7000);

                    IF temporalCounter_i1.done THEN 
                        (* Transition: '<S706>:15' *)
                        is_c59_ChiefMaster := ChiefMaster_IN_After_delay1;
                        (* Entry 'After_delay1': '<S706>:18' *)
                        (* '<S706>:18:3' out = In; *)
                        out := In;
                    ELSE 
                        (* '<S706>:20:3' out = false; *)
                        out := FALSE;
                    END_IF;

            END_CASE;

        END_IF;

        (* End of Chart: '<S702>/IMDOK_Input_Delay' *)
END_CASE;

END_FUNCTION_BLOCK

// Device/Application/Chart_Hysteresis_LowActive
FUNCTION_BLOCK Chart_Hysteresis_LowActive
VAR_INPUT
	ssMethodType: SINT;
	sSignal: REAL;
	boInitial_Value: BOOL;
	boValue_Activated: BOOL;
	boValue_Deactivated: BOOL;
	sLB: REAL;
	b_sUB: REAL;
END_VAR
VAR_OUTPUT
	boOutput: BOOL;
END_VAR
VAR
	is_active_c4_Library_DataProcessing_v1_1: USINT;
	is_c4_Library_DataProcessing_v1_1: USINT;
END_VAR



CASE ssMethodType OF
    SS_INITIALIZE: 
        is_active_c4_Library_DataProcessing_v1_1 := 0;
        is_c4_Library_DataProcessing_v1_1 := ChiefMaster_IN_NO_ACTIVE_CHILD_i2;
        boOutput := FALSE;
    SS_OUTPUT: 
        (* Chart: '<S410>/Chart_Hysteresis_LowActive' *)
        (* Gateway: Lib_Hysteresis_LowActive/Chart_Hysteresis_LowActive *)
        (* During: Lib_Hysteresis_LowActive/Chart_Hysteresis_LowActive *)

        IF is_active_c4_Library_DataProcessing_v1_1 = 0 THEN 
            (* Entry: Lib_Hysteresis_LowActive/Chart_Hysteresis_LowActive *)
            is_active_c4_Library_DataProcessing_v1_1 := 1;
            (* Entry Internal: Lib_Hysteresis_LowActive/Chart_Hysteresis_LowActive *)
            (* Transition: '<S411>:5' *)
            is_c4_Library_DataProcessing_v1_1 := ChiefMaster_IN_OFF_o;
            (* Entry 'OFF': '<S411>:8' *)
            (* '<S411>:8:3' boOutput= boInitial_Value; *)
            boOutput := boInitial_Value;
        ELSE 

            CASE is_c4_Library_DataProcessing_v1_1 OF
                ChiefMaster_IN_HighValue_a: 
                    (* During 'HighValue': '<S411>:4' *)
                    (* '<S411>:1:1' sf_internal_predicateOutput = sSignal>sUB; *)

                    IF sSignal > b_sUB THEN 
                        (* Transition: '<S411>:1' *)
                        is_c4_Library_DataProcessing_v1_1 := ChiefMaster_IN_LowValue_n;
                        (* Entry 'LowValue': '<S411>:2' *)
                        (* '<S411>:2:3' boOutput = boValue_Deactivated; *)
                        boOutput := boValue_Deactivated;
                    END_IF;

                ChiefMaster_IN_LowValue_n: 
                    (* During 'LowValue': '<S411>:2' *)
                    (* '<S411>:7:1' sf_internal_predicateOutput = sSignal<sLB; *)

                    IF sSignal < sLB THEN 
                        (* Transition: '<S411>:7' *)
                        is_c4_Library_DataProcessing_v1_1 := ChiefMaster_IN_HighValue_a;
                        (* Entry 'HighValue': '<S411>:4' *)
                        (* '<S411>:4:3' boOutput = boValue_Activated; *)
                        boOutput := boValue_Activated;
                    END_IF;

                ELSE
                    (* During 'OFF': '<S411>:8' *)
                    (* '<S411>:6:1' sf_internal_predicateOutput = sSignal>sUB; *)

                    IF sSignal > b_sUB THEN 
                        (* Transition: '<S411>:6' *)
                        is_c4_Library_DataProcessing_v1_1 := ChiefMaster_IN_LowValue_n;
                        (* Entry 'LowValue': '<S411>:2' *)
                        (* '<S411>:2:3' boOutput = boValue_Deactivated; *)
                        boOutput := boValue_Deactivated;
                    ELSE 
                        (* '<S411>:3:1' sf_internal_predicateOutput = sSignal<sLB; *)

                        IF sSignal < sLB THEN 
                            (* Transition: '<S411>:3' *)
                            is_c4_Library_DataProcessing_v1_1 := ChiefMaster_IN_HighValue_a;
                            (* Entry 'HighValue': '<S411>:4' *)
                            (* '<S411>:4:3' boOutput = boValue_Activated; *)
                            boOutput := boValue_Activated;
                        END_IF;

                    END_IF;

            END_CASE;

        END_IF;

        (* End of Chart: '<S410>/Chart_Hysteresis_LowActive' *)
END_CASE;

END_FUNCTION_BLOCK

// Device/Application/HVIL_Input_Delay
FUNCTION_BLOCK HVIL_Input_Delay
VAR_INPUT
	ssMethodType: SINT;
	HVIL_IN: BOOL;
	IP_HVIL_Delay_ms: USINT;
END_VAR
VAR_OUTPUT
	out: BOOL;
END_VAR
VAR
	is_active_c56_ChiefMaster: USINT;
	is_c56_ChiefMaster: USINT;
	temporalCounter_i1: PLC_CODER_TIMER;
END_VAR



CASE ssMethodType OF
    SS_INITIALIZE: 
        temporalCounter_i1(timerAction := 1, maxTime := 0);
        is_active_c56_ChiefMaster := 0;
        is_c56_ChiefMaster := ChiefMaster_IN_NO_ACTIVE_CHILD_cr;
        out := FALSE;
    SS_OUTPUT: 
        (* Chart: '<S384>/HVIL_Input_Delay' *)
        (* Gateway: ChiefMaster/Input Processing/HW Inputs/HVIL/HVIL_Input_Delay *)
        (* During: ChiefMaster/Input Processing/HW Inputs/HVIL/HVIL_Input_Delay *)

        IF is_active_c56_ChiefMaster = 0 THEN 
            (* Entry: ChiefMaster/Input Processing/HW Inputs/HVIL/HVIL_Input_Delay *)
            is_active_c56_ChiefMaster := 1;
            (* Entry Internal: ChiefMaster/Input Processing/HW Inputs/HVIL/HVIL_Input_Delay *)
            (* Transition: '<S399>:2' *)
            is_c56_ChiefMaster := ChiefMaster_IN_Initial_h;
            (* Entry 'Initial': '<S399>:1' *)
            (* '<S399>:1:3' out = HVIL_IN; *)
            out := HVIL_IN;
        ELSE 

            CASE is_c56_ChiefMaster OF
                ChiefMaster_IN_After_delay_c: 
                    (* During 'After_delay': '<S399>:4' *)
                    (* '<S399>:10:1' sf_internal_predicateOutput = HVIL_IN == false; *)

                    IF  NOT HVIL_IN THEN 
                        (* Transition: '<S399>:10' *)
                        is_c56_ChiefMaster := ChiefMaster_IN_Initial_h;
                        (* Entry 'Initial': '<S399>:1' *)
                        (* '<S399>:1:3' out = HVIL_IN; *)
                        out := FALSE;
                    ELSE 
                        (* '<S399>:4:3' out = HVIL_IN; *)
                        out := TRUE;
                    END_IF;

                ChiefMaster_IN_Delay_k: 
                    (* During 'Delay': '<S399>:3' *)
                    (* '<S399>:6:1' sf_internal_predicateOutput = after(IP_HVIL_Delay_ms, msec); *)
                    temporalCounter_i1(timerAction := 2, maxTime := USINT_TO_DINT(IP_HVIL_Delay_ms));

                    IF temporalCounter_i1.done THEN 
                        (* Transition: '<S399>:6' *)
                        is_c56_ChiefMaster := ChiefMaster_IN_After_delay_c;
                        (* Entry 'After_delay': '<S399>:4' *)
                        (* '<S399>:4:3' out = HVIL_IN; *)
                        out := HVIL_IN;
                    ELSE 
                        (* '<S399>:3:3' out = true; *)
                        out := TRUE;
                    END_IF;

                ELSE
                    (* During 'Initial': '<S399>:1' *)
                    (* '<S399>:5:1' sf_internal_predicateOutput = HVIL_IN == false; *)

                    IF  NOT HVIL_IN THEN 
                        (* Transition: '<S399>:5' *)
                        is_c56_ChiefMaster := ChiefMaster_IN_Delay_k;
                        temporalCounter_i1(timerAction := 1, maxTime := 0);
                        (* Entry 'Delay': '<S399>:3' *)
                        (* '<S399>:3:3' out = true; *)
                        out := TRUE;
                    ELSE 
                        (* '<S399>:1:3' out = HVIL_IN; *)
                        out := TRUE;
                    END_IF;

            END_CASE;

        END_IF;

        (* End of Chart: '<S384>/HVIL_Input_Delay' *)
END_CASE;

END_FUNCTION_BLOCK

// Device/Application/VoltageDetermination
FUNCTION_BLOCK VoltageDetermination
VAR_INPUT
	IP_sBMS_VtgInt_BB1: REAL;
	IP_sBMS_VtgInt_BB2: REAL;
	IP_sBMS_VtgInt_BB3: REAL;
	IP_boBMS_SDError_BB1: BOOL;
	IP_boBMS_SDError_BB2: BOOL;
	IP_boBMS_SDError_BB3: BOOL;
	IP_boBMS_Batt1_Availability: LREAL;
	IP_boBMS_Batt2_Availability: LREAL;
	IP_boBMS_Batt3_Availability: LREAL;
END_VAR
VAR_OUTPUT
	IT_u8BMS_BB_No_MaxVoltage: REAL;
	IT_u8BMS_BB_No_MinVoltage: REAL;
END_VAR
VAR
	rtb_AND7: BOOL;
	rtb_Switch4_o: LREAL;
	rtb_AND8: BOOL;
	rtb_Switch5_d: LREAL;
	rtb_AND9: BOOL;
	rtb_Switch6: LREAL;
	rtb_Switch7: REAL;
	rtb_Switch8: REAL;
	rtb_Switch9: REAL;
END_VAR


(* Logic: '<S705>/AND7' incorporates:
 *  Logic: '<S705>/NOT' *)
rtb_AND7 := ( NOT IP_boBMS_SDError_BB1) AND (IP_boBMS_Batt1_Availability <> 0.0);
(* Switch: '<S705>/Switch4' incorporates:
 *  Constant: '<S705>/Constant6' *)

IF rtb_AND7 THEN 
    rtb_Switch4_o := REAL_TO_LREAL(IP_sBMS_VtgInt_BB1);
ELSE 
    rtb_Switch4_o := 0.0;
END_IF;

(* End of Switch: '<S705>/Switch4' *)


(* Logic: '<S705>/AND8' incorporates:
 *  Logic: '<S705>/NOT1' *)
rtb_AND8 := ( NOT IP_boBMS_SDError_BB2) AND (IP_boBMS_Batt2_Availability <> 0.0);
(* Switch: '<S705>/Switch5' incorporates:
 *  Constant: '<S705>/Constant7' *)

IF rtb_AND8 THEN 
    rtb_Switch5_d := REAL_TO_LREAL(IP_sBMS_VtgInt_BB2);
ELSE 
    rtb_Switch5_d := 0.0;
END_IF;

(* End of Switch: '<S705>/Switch5' *)


(* Logic: '<S705>/AND9' incorporates:
 *  Logic: '<S705>/NOT2' *)
rtb_AND9 := ( NOT IP_boBMS_SDError_BB3) AND (IP_boBMS_Batt3_Availability <> 0.0);
(* Switch: '<S705>/Switch6' incorporates:
 *  Constant: '<S705>/Constant8' *)

IF rtb_AND9 THEN 
    rtb_Switch6 := REAL_TO_LREAL(IP_sBMS_VtgInt_BB3);
ELSE 
    rtb_Switch6 := 0.0;
END_IF;

(* End of Switch: '<S705>/Switch6' *)


(* Switch: '<S705>/Switch7' incorporates:
 *  Constant: '<S705>/Constant9'
 *  Constant: '<S709>/Constant'
 *  Logic: '<S705>/AND4'
 *  RelationalOperator: '<S709>/Compare' *)

IF (IP_sBMS_VtgInt_BB1 > 10.0) AND rtb_AND7 THEN 
    rtb_Switch7 := IP_sBMS_VtgInt_BB1;
ELSE 
    rtb_Switch7 := UINT_TO_REAL(Voltage_NA_UB);
END_IF;

(* End of Switch: '<S705>/Switch7' *)


(* Switch: '<S705>/Switch8' incorporates:
 *  Constant: '<S705>/Constant9'
 *  Constant: '<S710>/Constant'
 *  Logic: '<S705>/AND5'
 *  RelationalOperator: '<S710>/Compare' *)

IF (IP_sBMS_VtgInt_BB2 > 10.0) AND rtb_AND8 THEN 
    rtb_Switch8 := IP_sBMS_VtgInt_BB2;
ELSE 
    rtb_Switch8 := UINT_TO_REAL(Voltage_NA_UB);
END_IF;

(* End of Switch: '<S705>/Switch8' *)


(* Switch: '<S705>/Switch9' incorporates:
 *  Constant: '<S705>/Constant9'
 *  Constant: '<S711>/Constant'
 *  Logic: '<S705>/AND6'
 *  RelationalOperator: '<S711>/Compare' *)

IF (IP_sBMS_VtgInt_BB3 > 10.0) AND rtb_AND9 THEN 
    rtb_Switch9 := IP_sBMS_VtgInt_BB3;
ELSE 
    rtb_Switch9 := UINT_TO_REAL(Voltage_NA_UB);
END_IF;

(* End of Switch: '<S705>/Switch9' *)


(* Switch: '<S705>/Switch' incorporates:
 *  Constant: '<S705>/Constant'
 *  Logic: '<S705>/AND'
 *  Logic: '<S705>/AND1'
 *  RelationalOperator: '<S705>/GreaterThan'
 *  RelationalOperator: '<S705>/GreaterThan1'
 *  RelationalOperator: '<S705>/GreaterThan2'
 *  RelationalOperator: '<S705>/GreaterThan3'
 *  Switch: '<S705>/Switch1' *)

IF (rtb_Switch4_o >= rtb_Switch5_d) AND (rtb_Switch4_o >= rtb_Switch6) THEN 
    IT_u8BMS_BB_No_MaxVoltage := BattBox1_No;
ELSIF (rtb_Switch5_d >= rtb_Switch4_o) AND (rtb_Switch5_d >= rtb_Switch6) THEN 
    (* Switch: '<S705>/Switch1' incorporates:
     *  Constant: '<S705>/Constant1' *)
    IT_u8BMS_BB_No_MaxVoltage := BattBox2_No;
ELSE 
    (* Switch: '<S705>/Switch1' incorporates:
     *  Constant: '<S705>/Constant2' *)
    IT_u8BMS_BB_No_MaxVoltage := BattBox3_No;
END_IF;

(* End of Switch: '<S705>/Switch' *)


(* Switch: '<S705>/Switch2' incorporates:
 *  Constant: '<S705>/Constant'
 *  Logic: '<S705>/AND2'
 *  Logic: '<S705>/AND3'
 *  RelationalOperator: '<S705>/GreaterThan4'
 *  RelationalOperator: '<S705>/GreaterThan5'
 *  RelationalOperator: '<S705>/GreaterThan6'
 *  RelationalOperator: '<S705>/GreaterThan7'
 *  Switch: '<S705>/Switch3' *)

IF (rtb_Switch7 <= rtb_Switch8) AND (rtb_Switch7 <= rtb_Switch9) THEN 
    IT_u8BMS_BB_No_MinVoltage := BattBox1_No;
ELSIF (rtb_Switch8 <= rtb_Switch7) AND (rtb_Switch8 <= rtb_Switch9) THEN 
    (* Switch: '<S705>/Switch3' incorporates:
     *  Constant: '<S705>/Constant1' *)
    IT_u8BMS_BB_No_MinVoltage := BattBox2_No;
ELSE 
    (* Switch: '<S705>/Switch3' incorporates:
     *  Constant: '<S705>/Constant2' *)
    IT_u8BMS_BB_No_MinVoltage := BattBox3_No;
END_IF;

(* End of Switch: '<S705>/Switch2' *)

END_FUNCTION_BLOCK

// Device/Application/Receive
FUNCTION_BLOCK Receive
VAR_INPUT
END_VAR
VAR_OUTPUT
END_VAR
VAR

(* BMS *)
(*Batt1*)
	Actia_Batt1_Rx_140: CanRx;
	Actia_Batt1_Rx_100: CanRx;
	Actia_Batt1_Rx_600: CanRx;
	Actia_Batt1_Rx_500: CanRx;
	Actia_Batt1_Rx_520: CanRx;
	Actia_Batt1_Rx_560: CanRx;
(*Batt2*)
	Actia_Batt2_Rx_140: CanRx;
	Actia_Batt2_Rx_100: CanRx;
	Actia_Batt2_Rx_600: CanRx;
	Actia_Batt2_Rx_500: CanRx;
	Actia_Batt2_Rx_520: CanRx;
	Actia_Batt2_Rx_560: CanRx;
(*Batt3*)
	Actia_Batt3_Rx_140: CanRx;
	Actia_Batt3_Rx_100: CanRx;
	Actia_Batt3_Rx_600: CanRx;
	Actia_Batt3_Rx_500: CanRx;
	Actia_Batt3_Rx_520: CanRx;
	Actia_Batt3_Rx_560: CanRx;

(*LiBa*)
(*Batt1*)
	LB_Batt1_Rx_01: CanRx;
	LB_Batt1_Rx_02: CanRx;
	LB_Batt1_Rx_03: CanRx;
	LB_Batt1_Rx_04: CanRx;
	LB_Batt1_Rx_05: CanRx;
	LB_Batt1_Rx_06: CanRx;
	LB_Batt1_Rx_07: CanRx;
(*Batt2*)
	LB_Batt2_Rx_01: CanRx;
	LB_Batt2_Rx_02: CanRx;
	LB_Batt2_Rx_03: CanRx;
	LB_Batt2_Rx_04: CanRx;
	LB_Batt2_Rx_05: CanRx;
	LB_Batt2_Rx_06: CanRx;
	LB_Batt2_Rx_07: CanRx;
(*Batt3*)
	LB_Batt3_Rx_01: CanRx;
	LB_Batt3_Rx_02: CanRx;
	LB_Batt3_Rx_03: CanRx;
	LB_Batt3_Rx_04: CanRx;
	LB_Batt3_Rx_05: CanRx;
	LB_Batt3_Rx_06: CanRx;
	LB_Batt3_Rx_07: CanRx;
	
(*UDC*)
	UDC_Msg1: CanRx;

END_VAR


(**BMS**)

(*Actia*)
(*Box 1*)
(* BMS :0x140 *)
Actia_Batt1_Rx_140(iCAN:= ADR(GVL.gCan1),
				iCanId:= 16#140,
				iCanIdExtended:= FALSE,
				iTimeoutLimit:= T#1500MS,
				oByteCount=> ,
				oData=> GVL.C_Actia_BB1_MyStatus ,
				oNewData=> ,
				oCanTimeout=> GVL.C_Actia_BB1_MyStatus_Timeout,
				oReceiverId=> ,
				oTooManyReceivers=> );
				
(* BMS :0x100 *)
Actia_Batt1_Rx_100(iCAN:= ADR(GVL.gCan1),
				iCanId:= 16#100,
				iCanIdExtended:= FALSE,
				iTimeoutLimit:= T#1500MS,
				oByteCount=> ,
				oData=> GVL.C_Actia_BB1_Error ,
				oNewData=> ,
				oCanTimeout=> GVL.C_Actia_BB1_Error_Timeout,
				oReceiverId=> ,
				oTooManyReceivers=> );				
				
(* BMS :0x600 *)
Actia_Batt1_Rx_600(iCAN:= ADR(GVL.gCan1),
				iCanId:= 16#600,
				iCanIdExtended:= FALSE,
				iTimeoutLimit:= T#1500MS,
				oByteCount=> ,
				oData=> GVL.C_Actia_BB1_ADS_8 ,
				oNewData=> ,
				oCanTimeout=> GVL.C_Actia_BB1_ADS_8_Timeout,
				oReceiverId=> ,
				oTooManyReceivers=> );
				
(* BMS :0x500 *)
Actia_Batt1_Rx_500(iCAN:= ADR(GVL.gCan1),
				iCanId:= 16#500,
				iCanIdExtended:= FALSE,
				iTimeoutLimit:= T#1500MS,
				oByteCount=> ,
				oData=> GVL.C_Actia_BB1_ADS_0,
				oNewData=> ,
				oCanTimeout=> GVL.C_Actia_BB1_ADS_0_Timeout,
				oReceiverId=> ,
				oTooManyReceivers=> );				
				
(* BMS :0x520 *)
Actia_Batt1_Rx_520(iCAN:= ADR(GVL.gCan1),
				iCanId:= 16#520,
				iCanIdExtended:= FALSE,
				iTimeoutLimit:= T#1500MS,
				oByteCount=> ,
				oData=> GVL.C_Actia_BB1_ADS_1 ,
				oNewData=> ,
				oCanTimeout=> GVL.C_Actia_BB1_ADS_1_Timeout,
				oReceiverId=> ,
				oTooManyReceivers=> );

(* BMS :0x560 *)
Actia_Batt1_Rx_560(iCAN:= ADR(GVL.gCan1),
				iCanId:= 16#560,
				iCanIdExtended:= FALSE,
				iTimeoutLimit:= T#1500MS,
				oByteCount=> ,
				oData=> GVL.C_Actia_BB1_ADS_3 ,
				oNewData=> ,
				oCanTimeout=> GVL.C_Actia_BB1_ADS_3_Timeout,
				oReceiverId=> ,
				oTooManyReceivers=> );

(*Box 2*)
(* BMS :0x140 *)
Actia_Batt2_Rx_140(iCAN:= ADR(GVL.gCan2),
				iCanId:= 16#140,
				iCanIdExtended:= FALSE,
				iTimeoutLimit:= T#1500MS,
				oByteCount=> ,
				oData=> GVL.C_Actia_BB2_MyStatus ,
				oNewData=> ,
				oCanTimeout=> GVL.C_Actia_BB2_MyStatus_Timeout,
				oReceiverId=> ,
				oTooManyReceivers=> );
				
(* BMS :0x100 *)
Actia_Batt2_Rx_100(iCAN:= ADR(GVL.gCan2),
				iCanId:= 16#100,
				iCanIdExtended:= FALSE,
				iTimeoutLimit:= T#1500MS,
				oByteCount=> ,
				oData=> GVL.C_Actia_BB2_Error ,
				oNewData=> ,
				oCanTimeout=> GVL.C_Actia_BB2_Error_Timeout,
				oReceiverId=> ,
				oTooManyReceivers=> );				
				
(* BMS :0x600 *)
Actia_Batt2_Rx_600(iCAN:= ADR(GVL.gCan2),
				iCanId:= 16#600,
				iCanIdExtended:= FALSE,
				iTimeoutLimit:= T#1500MS,
				oByteCount=> ,
				oData=> GVL.C_Actia_BB2_ADS_8 ,
				oNewData=> ,
				oCanTimeout=> GVL.C_Actia_BB2_ADS_8_Timeout,
				oReceiverId=> ,
				oTooManyReceivers=> );
				
(* BMS :0x500 *)
Actia_Batt2_Rx_500(iCAN:= ADR(GVL.gCan2),
				iCanId:= 16#500,
				iCanIdExtended:= FALSE,
				iTimeoutLimit:= T#1500MS,
				oByteCount=> ,
				oData=> GVL.C_Actia_BB2_ADS_0,
				oNewData=> ,
				oCanTimeout=> GVL.C_Actia_BB2_ADS_0_Timeout,
				oReceiverId=> ,
				oTooManyReceivers=> );	
				
(* BMS :0x520 *)
Actia_Batt2_Rx_520(iCAN:= ADR(GVL.gCan2),
				iCanId:= 16#520,
				iCanIdExtended:= FALSE,
				iTimeoutLimit:= T#1500MS,
				oByteCount=> ,
				oData=> GVL.C_Actia_BB2_ADS_1 ,
				oNewData=> ,
				oCanTimeout=> GVL.C_Actia_BB2_ADS_1_Timeout,
				oReceiverId=> ,
				oTooManyReceivers=> );

(* BMS :0x560 *)
Actia_Batt2_Rx_560(iCAN:= ADR(GVL.gCan2),
				iCanId:= 16#560,
				iCanIdExtended:= FALSE,
				iTimeoutLimit:= T#1500MS,
				oByteCount=> ,
				oData=> GVL.C_Actia_BB2_ADS_3 ,
				oNewData=> ,
				oCanTimeout=> GVL.C_Actia_BB2_ADS_3_Timeout,
				oReceiverId=> ,
				oTooManyReceivers=> );

(*Box 3*)
(* BMS :0x140 *)
Actia_Batt3_Rx_140(iCAN:= ADR(GVL.gCan3),
				iCanId:= 16#140,
				iCanIdExtended:= FALSE,
				iTimeoutLimit:= T#1500MS,
				oByteCount=> ,
				oData=> GVL.C_Actia_BB3_MyStatus ,
				oNewData=> ,
				oCanTimeout=> GVL.C_Actia_BB3_MyStatus_Timeout,
				oReceiverId=> ,
				oTooManyReceivers=> );
				
(* BMS :0x100 *)
Actia_Batt3_Rx_100(iCAN:= ADR(GVL.gCan3),
				iCanId:= 16#100,
				iCanIdExtended:= FALSE,
				iTimeoutLimit:= T#1500MS,
				oByteCount=> ,
				oData=> GVL.C_Actia_BB3_Error ,
				oNewData=> ,
				oCanTimeout=> GVL.C_Actia_BB3_Error_Timeout,
				oReceiverId=> ,
				oTooManyReceivers=> );				
				
(* BMS :0x600 *)
Actia_Batt3_Rx_600(iCAN:= ADR(GVL.gCan3),
				iCanId:= 16#600,
				iCanIdExtended:= FALSE,
				iTimeoutLimit:= T#1500MS,
				oByteCount=> ,
				oData=> GVL.C_Actia_BB3_ADS_8 ,
				oNewData=> ,
				oCanTimeout=> GVL.C_Actia_BB3_ADS_8_Timeout,
				oReceiverId=> ,
				oTooManyReceivers=> );
				
(* BMS :0x500 *)
Actia_Batt3_Rx_500(iCAN:= ADR(GVL.gCan3),
				iCanId:= 16#500,
				iCanIdExtended:= FALSE,
				iTimeoutLimit:= T#1500MS,
				oByteCount=> ,
				oData=> GVL.C_Actia_BB3_ADS_0,
				oNewData=> ,
				oCanTimeout=> GVL.C_Actia_BB3_ADS_0_Timeout,
				oReceiverId=> ,
				oTooManyReceivers=> );	
				
(* BMS :0x520 *)
Actia_Batt3_Rx_520(iCAN:= ADR(GVL.gCan3),
				iCanId:= 16#520,
				iCanIdExtended:= FALSE,
				iTimeoutLimit:= T#1500MS,
				oByteCount=> ,
				oData=> GVL.C_Actia_BB3_ADS_1 ,
				oNewData=> ,
				oCanTimeout=> GVL.C_Actia_BB3_ADS_1_Timeout,
				oReceiverId=> ,
				oTooManyReceivers=> );

(* BMS :0x560 *)
Actia_Batt3_Rx_560(iCAN:= ADR(GVL.gCan3),
				iCanId:= 16#560,
				iCanIdExtended:= FALSE,
				iTimeoutLimit:= T#1500MS,
				oByteCount=> ,
				oData=> GVL.C_Actia_BB3_ADS_3 ,
				oNewData=> ,
				oCanTimeout=> GVL.C_Actia_BB3_ADS_3_Timeout,
				oReceiverId=> ,
				oTooManyReceivers=> );
				
(*LiBa*)
(*Batt1*)
LB_Batt1_Rx_01(
	iCAN:= ADR(GVL.gCan1),
	iCanId:= 16#18FF03F3,
	iCanIdExtended:= TRUE,
	iTimeoutLimit:= T#1000MS,
	oByteCount=> ,
	oData=> GVL.C_LB_Batt1_CellVoltage01,
	oNewData=> ,
	oCanTimeout=> GVL.C_LB_Batt1_CellVoltage01_Timeout,
	oReceiverId=> ,
	oTooManyReceivers=> );

LB_Batt1_Rx_02(
	iCAN:= ADR(GVL.gCan1),
	iCanId:= 16#18FF04F3,
	iCanIdExtended:= TRUE,
	iTimeoutLimit:= T#1000MS,
	oByteCount=> ,
	oData=> GVL.C_LB_Batt1_CellVoltage02,
	oNewData=> ,
	oCanTimeout=> GVL.C_LB_Batt1_CellVoltage02_Timeout,
	oReceiverId=> ,
	oTooManyReceivers=> );

LB_Batt1_Rx_03(
	iCAN:= ADR(GVL.gCan1),
	iCanId:= 16#18FF05F3,
	iCanIdExtended:= TRUE,
	iTimeoutLimit:= T#1000MS,
	oByteCount=> ,
	oData=> GVL.C_LB_Batt1_CellTemperature,
	oNewData=> ,
	oCanTimeout=> GVL.C_LB_Batt1_CellTemperature_Timeout,
	oReceiverId=> ,
	oTooManyReceivers=> );

LB_Batt1_Rx_04(
	iCAN:= ADR(GVL.gCan1),
	iCanId:= 16#18FF06F3,
	iCanIdExtended:= TRUE,
	iTimeoutLimit:= T#1000MS,
	oByteCount=> ,
	oData=> GVL.C_LB_Batt1_InsulationMonitor,
	oNewData=> ,
	oCanTimeout=> GVL.C_LB_Batt1_InsulationMonitor_Timeout,
	oReceiverId=> ,
	oTooManyReceivers=> );

LB_Batt1_Rx_05(
	iCAN:= ADR(GVL.gCan1),
	iCanId:= 16#18FF01F3,
	iCanIdExtended:= TRUE,
	iTimeoutLimit:= T#1000MS,
	oByteCount=> ,
	oData=> GVL.C_LB_Batt1_Status01,
	oNewData=> ,
	oCanTimeout=> GVL.C_LB_Batt1_Status01_Timeout,
	oReceiverId=> ,
	oTooManyReceivers=> );

LB_Batt1_Rx_06(
	iCAN:= ADR(GVL.gCan1),
	iCanId:= 16#18FF02F3,
	iCanIdExtended:= TRUE,
	iTimeoutLimit:= T#1000MS,
	oByteCount=> ,
	oData=> GVL.C_LB_Batt1_Status02,
	oNewData=> ,
	oCanTimeout=> GVL.C_LB_Batt1_Status02_Timeout,
	oReceiverId=> ,
	oTooManyReceivers=> );

LB_Batt1_Rx_07(
	iCAN:= ADR(GVL.gCan1),
	iCanId:= 16#18FF07F3,
	iCanIdExtended:= TRUE,
	iTimeoutLimit:= T#1000MS,
	oByteCount=> ,
	oData=> GVL.C_LB_Batt1_Status03,
	oNewData=> ,
	oCanTimeout=> GVL.C_LB_Batt1_Status03_Timeout,
	oReceiverId=> ,
	oTooManyReceivers=> );
				
(*Batt2*)
LB_Batt2_Rx_01(
	iCAN:= ADR(GVL.gCan2),
	iCanId:= 16#18FF03F3,
	iCanIdExtended:= TRUE,
	iTimeoutLimit:= T#1000MS,
	oByteCount=> ,
	oData=> GVL.C_LB_Batt2_CellVoltage01,
	oNewData=> ,
	oCanTimeout=> GVL.C_LB_Batt2_CellVoltage01_Timeout,
	oReceiverId=> ,
	oTooManyReceivers=> );

LB_Batt2_Rx_02(
	iCAN:= ADR(GVL.gCan2),
	iCanId:= 16#18FF04F3,
	iCanIdExtended:= TRUE,
	iTimeoutLimit:= T#1000MS,
	oByteCount=> ,
	oData=> GVL.C_LB_Batt2_CellVoltage02,
	oNewData=> ,
	oCanTimeout=> GVL.C_LB_Batt2_CellVoltage02_Timeout,
	oReceiverId=> ,
	oTooManyReceivers=> );

LB_Batt2_Rx_03(
	iCAN:= ADR(GVL.gCan2),
	iCanId:= 16#18FF05F3,
	iCanIdExtended:= TRUE,
	iTimeoutLimit:= T#1000MS,
	oByteCount=> ,
	oData=> GVL.C_LB_Batt2_CellTemperature,
	oNewData=> ,
	oCanTimeout=> GVL.C_LB_Batt2_CellTemperature_Timeout,
	oReceiverId=> ,
	oTooManyReceivers=> );

LB_Batt2_Rx_04(
	iCAN:= ADR(GVL.gCan2),
	iCanId:= 16#18FF06F3,
	iCanIdExtended:= TRUE,
	iTimeoutLimit:= T#1000MS,
	oByteCount=> ,
	oData=> GVL.C_LB_Batt2_InsulationMonitor,
	oNewData=> ,
	oCanTimeout=> GVL.C_LB_Batt2_InsulationMonitor_Timeout,
	oReceiverId=> ,
	oTooManyReceivers=> );

LB_Batt2_Rx_05(
	iCAN:= ADR(GVL.gCan2),
	iCanId:= 16#18FF01F3,
	iCanIdExtended:= TRUE,
	iTimeoutLimit:= T#1000MS,
	oByteCount=> ,
	oData=> GVL.C_LB_Batt2_Status01,
	oNewData=> ,
	oCanTimeout=> GVL.C_LB_Batt2_Status01_Timeout,
	oReceiverId=> ,
	oTooManyReceivers=> );

LB_Batt2_Rx_06(
	iCAN:= ADR(GVL.gCan2),
	iCanId:= 16#18FF02F3,
	iCanIdExtended:= TRUE,
	iTimeoutLimit:= T#1000MS,
	oByteCount=> ,
	oData=> GVL.C_LB_Batt2_Status02,
	oNewData=> ,
	oCanTimeout=> GVL.C_LB_Batt2_Status02_Timeout,
	oReceiverId=> ,
	oTooManyReceivers=> );

LB_Batt2_Rx_07(
	iCAN:= ADR(GVL.gCan2),
	iCanId:= 16#18FF07F3,
	iCanIdExtended:= TRUE,
	iTimeoutLimit:= T#1000MS,
	oByteCount=> ,
	oData=> GVL.C_LB_Batt2_Status03,
	oNewData=> ,
	oCanTimeout=> GVL.C_LB_Batt2_Status03_Timeout,
	oReceiverId=> ,
	oTooManyReceivers=> );
	
(*Batt3*)
LB_Batt3_Rx_01(
	iCAN:= ADR(GVL.gCan3),
	iCanId:= 16#18FF03F3,
	iCanIdExtended:= TRUE,
	iTimeoutLimit:= T#1000MS,
	oByteCount=> ,
	oData=> GVL.C_LB_Batt3_CellVoltage01,
	oNewData=> ,
	oCanTimeout=> GVL.C_LB_Batt3_CellVoltage01_Timeout,
	oReceiverId=> ,
	oTooManyReceivers=> );

LB_Batt3_Rx_02(
	iCAN:= ADR(GVL.gCan3),
	iCanId:= 16#18FF04F3,
	iCanIdExtended:= TRUE,
	iTimeoutLimit:= T#1000MS,
	oByteCount=> ,
	oData=> GVL.C_LB_Batt3_CellVoltage02,
	oNewData=> ,
	oCanTimeout=> GVL.C_LB_Batt3_CellVoltage02_Timeout,
	oReceiverId=> ,
	oTooManyReceivers=> );

LB_Batt3_Rx_03(
	iCAN:= ADR(GVL.gCan3),
	iCanId:= 16#18FF05F3,
	iCanIdExtended:= TRUE,
	iTimeoutLimit:= T#1000MS,
	oByteCount=> ,
	oData=> GVL.C_LB_Batt3_CellTemperature,
	oNewData=> ,
	oCanTimeout=> GVL.C_LB_Batt3_CellTemperature_Timeout,
	oReceiverId=> ,
	oTooManyReceivers=> );

LB_Batt3_Rx_04(
	iCAN:= ADR(GVL.gCan3),
	iCanId:= 16#18FF06F3,
	iCanIdExtended:= TRUE,
	iTimeoutLimit:= T#1000MS,
	oByteCount=> ,
	oData=> GVL.C_LB_Batt3_InsulationMonitor,
	oNewData=> ,
	oCanTimeout=> GVL.C_LB_Batt3_InsulationMonitor_Timeout,
	oReceiverId=> ,
	oTooManyReceivers=> );

LB_Batt3_Rx_05(
	iCAN:= ADR(GVL.gCan3),
	iCanId:= 16#18FF01F3,
	iCanIdExtended:= TRUE,
	iTimeoutLimit:= T#1000MS,
	oByteCount=> ,
	oData=> GVL.C_LB_Batt3_Status01,
	oNewData=> ,
	oCanTimeout=> GVL.C_LB_Batt3_Status01_Timeout,
	oReceiverId=> ,
	oTooManyReceivers=> );

LB_Batt3_Rx_06(
	iCAN:= ADR(GVL.gCan3),
	iCanId:= 16#18FF02F3,
	iCanIdExtended:= TRUE,
	iTimeoutLimit:= T#1000MS,
	oByteCount=> ,
	oData=> GVL.C_LB_Batt3_Status02,
	oNewData=> ,
	oCanTimeout=> GVL.C_LB_Batt3_Status02_Timeout,
	oReceiverId=> ,
	oTooManyReceivers=> );

LB_Batt3_Rx_07(
	iCAN:= ADR(GVL.gCan3),
	iCanId:= 16#18FF07F3,
	iCanIdExtended:= TRUE,
	iTimeoutLimit:= T#1000MS,
	oByteCount=> ,
	oData=> GVL.C_LB_Batt3_Status03,
	oNewData=> ,
	oCanTimeout=> GVL.C_LB_Batt3_Status03_Timeout,
	oReceiverId=> ,
	oTooManyReceivers=> );	
	
(*UDC*)

UDC_Msg1(
	iCAN:= ADR(GVL.gCan0),
	iCanId:=  16#299,
	iCanIdExtended:= FALSE,
	iTimeoutLimit:= T#1500MS,
	oByteCount=> ,
	oData=> GVL.C_UDC_Msg1,
	oNewData=> ,
	oCanTimeout=> GVL.C_UDC_Msg1_Timeout,
	oReceiverId=> , 
	oTooManyReceivers=> );

END_FUNCTION_BLOCK

// Device/Application/Transmit
FUNCTION_BLOCK Transmit
VAR_INPUT
END_VAR
VAR_OUTPUT
END_VAR
VAR

(* BattBox *)
	Actia_Control_Batt1: CanTx;
	Actia_Control_Batt2: CanTx;
	Actia_Control_Batt3: CanTx;

	LiBa_Control_Batt1: CanTx;
	LiBa_Control_Batt2: CanTx;
	LiBa_Control_Batt3: CanTx;

(*Chief Master*)
	Chief_Master_Msg1: CanTx;
	Chief_Master_Msg2: CanTx;
	Chief_Master_Msg3: CanTx;
	Chief_Master_Msg4: CanTx;
	Chief_Master_Msg5: CanTx;
	Chief_Master_Msg6: CanTx;
	Chief_Master_Msg7: CanTx;
	Chief_Master_Msg8: CanTx;
	Chief_Master_Msg9: CanTx;
	Chief_Master_Msg10: CanTx;
	Chief_Master_Msg11: CanTx;
	Chief_Master_Msg12: CanTx;
	Chief_Master_Msg13: CanTx;
	Chief_Master_Msg14: CanTx;
	Chief_Master_Msg15: CanTx;

END_VAR

(*Actia*)
Actia_Control_Batt1(
				iEnable:= TRUE, 
				iCAN:= ADR(GVL.gCan1), 
				iForceSend:= FALSE, 
				iTransmitRate:= T#100MS, 
				iCanId:= 16#80, 
				iCanIdExtended:= FALSE, 
				iByteCount:= 8, 
				iData:= GVL.C_Actia_Control_Batt1, 
				oTransmitterId=> , 
				oTooManyTransmitters=> , 
				oMsgSent=> );
				
Actia_Control_Batt2(
				iEnable:= TRUE, 
				iCAN:= ADR(GVL.gCan2), 
				iForceSend:= FALSE, 
				iTransmitRate:= T#100MS, 
				iCanId:= 16#80, 
				iCanIdExtended:= FALSE, 
				iByteCount:= 8, 
				iData:= GVL.C_Actia_Control_Batt2, 
				oTransmitterId=> , 
				oTooManyTransmitters=> , 
				oMsgSent=> );
				
Actia_Control_Batt3(
				iEnable:= TRUE, 
				iCAN:= ADR(GVL.gCan3), 
				iForceSend:= FALSE, 
				iTransmitRate:= T#100MS, 
				iCanId:= 16#80, 
				iCanIdExtended:= FALSE, 
				iByteCount:= 8, 
				iData:= GVL.C_Actia_Control_Batt3, 
				oTransmitterId=> , 
				oTooManyTransmitters=> , 
				oMsgSent=> );				
				
(*LiBa*)
LiBa_Control_Batt1(
				iEnable:= TRUE,
				iCAN:= ADR(GVL.gCan1),
				iForceSend:= FALSE,
				iTransmitRate:= T#100MS,
				iCanId:= 16#18FFF369,
				iCanIdExtended:= TRUE,
				iByteCount:= 8,
				iData:= GVL.C_LiBa_OperationRequest_Batt1,
				oTransmitterId=> ,
				oTooManyTransmitters=> ,
				oMsgSent=> );

LiBa_Control_Batt2(
				iEnable:= TRUE,
				iCAN:= ADR(GVL.gCan2),
				iForceSend:= FALSE,
				iTransmitRate:= T#100MS,
				iCanId:= 16#18FFF369,
				iCanIdExtended:= TRUE,
				iByteCount:= 8,
				iData:= GVL.C_LiBa_OperationRequest_Batt2,
				oTransmitterId=> ,
				oTooManyTransmitters=> ,
				oMsgSent=> );

LiBa_Control_Batt3(
				iEnable:= TRUE,
				iCAN:= ADR(GVL.gCan3),
				iForceSend:= FALSE,
				iTransmitRate:= T#100MS,
				iCanId:= 16#18FFF369,
				iCanIdExtended:= TRUE,
				iByteCount:= 8,
				iData:= GVL.C_LiBa_OperationRequest_Batt3,
				oTransmitterId=> ,
				oTooManyTransmitters=> ,
				oMsgSent=> );

(*Chief Master*)				
Chief_Master_Msg1(
				iEnable:= TRUE, 
				iCAN:= ADR(GVL.gCan0), 
				iForceSend:= FALSE, 
				iTransmitRate:= T#100MS, 
				iCanId:= 16#85, 
				iCanIdExtended:= FALSE, 
				iByteCount:= 8, 
				iData:= GVL.C_Chief_Master_Msg1, 
				oTransmitterId=> , 
				oTooManyTransmitters=> , 
				oMsgSent=> );

Chief_Master_Msg2(
				iEnable:= TRUE, 
				iCAN:= ADR(GVL.gCan0), 
				iForceSend:= FALSE, 
				iTransmitRate:= T#100MS, 
				iCanId:= 16#86, 
				iCanIdExtended:= FALSE, 
				iByteCount:= 8, 
				iData:= GVL.C_Chief_Master_Msg2, 
				oTransmitterId=> , 
				oTooManyTransmitters=> , 
				oMsgSent=> );
				
Chief_Master_Msg3(
				iEnable:= TRUE, 
				iCAN:= ADR(GVL.gCan0), 
				iForceSend:= FALSE, 
				iTransmitRate:= T#100MS, 
				iCanId:= 16#87, 
				iCanIdExtended:= FALSE, 
				iByteCount:= 8, 
				iData:= GVL.C_Chief_Master_Msg3, 
				oTransmitterId=> , 
				oTooManyTransmitters=> , 
				oMsgSent=> );

Chief_Master_Msg4(
				iEnable:= TRUE, 
				iCAN:= ADR(GVL.gCan0), 
				iForceSend:= FALSE, 
				iTransmitRate:= T#100MS, 
				iCanId:= 16#88, 
				iCanIdExtended:= FALSE, 
				iByteCount:= 8, 
				iData:= GVL.C_Chief_Master_Msg4, 
				oTransmitterId=> , 
				oTooManyTransmitters=> , 
				oMsgSent=> );

Chief_Master_Msg5(
				iEnable:= TRUE, 
				iCAN:= ADR(GVL.gCan0), 
				iForceSend:= FALSE, 
				iTransmitRate:= T#1000MS, 
				iCanId:= 16#89, 
				iCanIdExtended:= FALSE, 
				iByteCount:= 8, 
				iData:= GVL.C_Chief_Master_Msg5, 
				oTransmitterId=> , 
				oTooManyTransmitters=> , 
				oMsgSent=> );

Chief_Master_Msg6(
				iEnable:= TRUE, 
				iCAN:= ADR(GVL.gCan0), 
				iForceSend:= FALSE, 
				iTransmitRate:= T#100MS, 
				iCanId:= 16#90, 
				iCanIdExtended:= FALSE, 
				iByteCount:= 8, 
				iData:= GVL.C_Chief_Master_Msg6, 
				oTransmitterId=> , 
				oTooManyTransmitters=> , 
				oMsgSent=> );
				
Chief_Master_Msg7(
				iEnable:= TRUE, 
				iCAN:= ADR(GVL.gCan0), 
				iForceSend:= FALSE, 
				iTransmitRate:= T#100MS, 
				iCanId:= 16#91, 
				iCanIdExtended:= FALSE, 
				iByteCount:= 8, 
				iData:= GVL.C_Chief_Master_Msg7, 
				oTransmitterId=> , 
				oTooManyTransmitters=> , 
				oMsgSent=> );

Chief_Master_Msg8(
				iEnable:= TRUE, 
				iCAN:= ADR(GVL.gCan0), 
				iForceSend:= FALSE, 
				iTransmitRate:= T#1000MS, 
				iCanId:= 16#92, 
				iCanIdExtended:= FALSE, 
				iByteCount:= 8, 
				iData:= GVL.C_Chief_Master_Msg8, 
				oTransmitterId=> , 
				oTooManyTransmitters=> , 
				oMsgSent=> );								
				
Chief_Master_Msg9(
				iEnable:= TRUE, 
				iCAN:= ADR(GVL.gCan0), 
				iForceSend:= FALSE, 
				iTransmitRate:= T#1000MS, 
				iCanId:= 16#93, 
				iCanIdExtended:= FALSE, 
				iByteCount:= 8, 
				iData:= GVL.C_Chief_Master_Msg9, 
				oTransmitterId=> , 
				oTooManyTransmitters=> , 
				oMsgSent=> );

Chief_Master_Msg10(
				iEnable:= TRUE, 
				iCAN:= ADR(GVL.gCan0), 
				iForceSend:= FALSE, 
				iTransmitRate:= T#100MS, 
				iCanId:= 16#94, 
				iCanIdExtended:= FALSE, 
				iByteCount:= 8, 
				iData:= GVL.C_Chief_Master_Msg10, 
				oTransmitterId=> , 
				oTooManyTransmitters=> , 
				oMsgSent=> );
				
Chief_Master_Msg11(
				iEnable:= TRUE, 
				iCAN:= ADR(GVL.gCan0), 
				iForceSend:= FALSE, 
				iTransmitRate:= T#1000MS, 
				iCanId:= 16#95, 
				iCanIdExtended:= FALSE, 
				iByteCount:= 8, 
				iData:= GVL.C_Chief_Master_Msg11, 
				oTransmitterId=> , 
				oTooManyTransmitters=> , 
				oMsgSent=> );

Chief_Master_Msg12(
				iEnable:= TRUE, 
				iCAN:= ADR(GVL.gCan0), 
				iForceSend:= FALSE, 
				iTransmitRate:= T#1000MS, 
				iCanId:= 16#96, 
				iCanIdExtended:= FALSE, 
				iByteCount:= 8, 
				iData:= GVL.C_Chief_Master_Msg12, 
				oTransmitterId=> , 
				oTooManyTransmitters=> , 
				oMsgSent=> );	
				
Chief_Master_Msg13(
				iEnable:= TRUE, 
				iCAN:= ADR(GVL.gCan0), 
				iForceSend:= FALSE, 
				iTransmitRate:= T#100MS, 
				iCanId:= 16#97, 
				iCanIdExtended:= FALSE, 
				iByteCount:= 8, 
				iData:= GVL.C_Chief_Master_Msg13, 
				oTransmitterId=> , 
				oTooManyTransmitters=> , 
				oMsgSent=> );
				
Chief_Master_Msg14(
				iEnable:= TRUE, 
				iCAN:= ADR(GVL.gCan0), 
				iForceSend:= FALSE, 
				iTransmitRate:= T#1000MS, 
				iCanId:= 16#98, 
				iCanIdExtended:= FALSE, 
				iByteCount:= 8, 
				iData:= GVL.C_Chief_Master_Msg14, 
				oTransmitterId=> , 
				oTooManyTransmitters=> , 
				oMsgSent=> );

Chief_Master_Msg15(
				iEnable:= TRUE, 
				iCAN:= ADR(GVL.gCan0), 
				iForceSend:= FALSE, 
				iTransmitRate:= T#1000MS, 
				iCanId:= 16#99, 
				iCanIdExtended:= FALSE, 
				iByteCount:= 8, 
				iData:= GVL.C_Chief_Master_Msg15, 
				oTransmitterId=> , 
				oTooManyTransmitters=> , 
				oMsgSent=> );

END_FUNCTION_BLOCK

// Device/Application/Chart_j
FUNCTION_BLOCK Chart_j
VAR_INPUT
	ssMethodType: SINT;
	In: LREAL;
	b_n: LREAL;
END_VAR
VAR_OUTPUT
	Out: BOOL;
END_VAR
VAR
	is_c10_ChiefMaster: USINT;
	temporalCounter_i1: PLC_CODER_TIMER;
	is_active_c10_ChiefMaster: USINT;
END_VAR



CASE ssMethodType OF
    SS_INITIALIZE: 
        temporalCounter_i1(timerAction := 1, maxTime := 0);
        is_active_c10_ChiefMaster := 0;
        is_c10_ChiefMaster := ChiefMaster_IN_NO_ACTIVE_CHILD_a4;
        Out := FALSE;
    SS_OUTPUT: 
        (* Chart: '<S78>/Chart' *)
        (* Gateway: ChiefMaster/Flow Logic/Reset/Reset_Req/Subsystem1/Chart *)
        (* During: ChiefMaster/Flow Logic/Reset/Reset_Req/Subsystem1/Chart *)

        IF is_active_c10_ChiefMaster = 0 THEN 
            (* Entry: ChiefMaster/Flow Logic/Reset/Reset_Req/Subsystem1/Chart *)
            is_active_c10_ChiefMaster := 1;
            (* Entry Internal: ChiefMaster/Flow Logic/Reset/Reset_Req/Subsystem1/Chart *)
            (* Transition: '<S84>:3' *)
            is_c10_ChiefMaster := ChiefMaster_IN_Default_m;
            (* Entry 'Default': '<S84>:2' *)
            (* '<S84>:2:2' Out = false *)
            Out := FALSE;
        ELSE 

            CASE is_c10_ChiefMaster OF
                ChiefMaster_IN_Default_m: 
                    (* During 'Default': '<S84>:2' *)
                    (* '<S84>:6:1' sf_internal_predicateOutput = In == 2; *)

                    IF In = 2.0 THEN 
                        (* Transition: '<S84>:6' *)
                        is_c10_ChiefMaster := ChiefMaster_IN_Delay;
                        temporalCounter_i1(timerAction := 1, maxTime := 0);
                        (* Entry 'Delay': '<S84>:5' *)
                        (* '<S84>:5:2' Out = false *)
                        Out := FALSE;
                    ELSE 
                        (* '<S84>:2:2' Out = false *)
                        Out := FALSE;
                    END_IF;

                ChiefMaster_IN_Delay: 
                    (* During 'Delay': '<S84>:5' *)
                    (* '<S84>:12:1' sf_internal_predicateOutput = after(n,sec); *)
                    temporalCounter_i1(timerAction := 2, maxTime := TRUNC(b_n * 1000.0));

                    IF temporalCounter_i1.done THEN 
                        (* Transition: '<S84>:12' *)
                        is_c10_ChiefMaster := b_ChiefMaster_IN_Delay1;
                        (* Entry 'Delay1': '<S84>:11' *)
                        (* '<S84>:11:2' Out = true *)
                        Out := TRUE;
                    ELSE 
                        (* '<S84>:13:1' sf_internal_predicateOutput = In == 1 ||... *)
                        (* '<S84>:13:2' In == 3; *)

                        IF (In = 1.0) OR (In = 3.0) THEN 
                            (* Transition: '<S84>:13' *)
                            is_c10_ChiefMaster := ChiefMaster_IN_Default_m;
                            (* Entry 'Default': '<S84>:2' *)
                            (* '<S84>:2:2' Out = false *)
                            Out := FALSE;
                        ELSE 
                            (* '<S84>:5:2' Out = false *)
                            Out := FALSE;
                        END_IF;

                    END_IF;

                ELSE
                    (* During 'Delay1': '<S84>:11' *)
                    (* '<S84>:14:1' sf_internal_predicateOutput = In == 3; *)

                    IF In = 3.0 THEN 
                        (* Transition: '<S84>:14' *)
                        is_c10_ChiefMaster := ChiefMaster_IN_Default_m;
                        (* Entry 'Default': '<S84>:2' *)
                        (* '<S84>:2:2' Out = false *)
                        Out := FALSE;
                    ELSE 
                        (* '<S84>:11:2' Out = true *)
                        Out := TRUE;
                    END_IF;

            END_CASE;

        END_IF;

        (* End of Chart: '<S78>/Chart' *)
END_CASE;

END_FUNCTION_BLOCK
